LIN {X 0,Y 538.147,Z 457.446,A -85,B 0,C 180,E1 -4137.754,E2 -4137.754} C_VEL
LIN {X 0,Y 538.174,Z 457.449,A -85,B 0,C 180,E1 -4140.748,E2 -4140.748} C_VEL
LIN {X 0,Y 538.129,Z 457.451,A -85,B 0,C 180,E1 -4142.994,E2 -4142.994} C_VEL
LIN {X 0,Y 538.104,Z 457.452,A -85,B 0,C 180,E1 -4145.997,E2 -4145.997} C_VEL
LIN {X 0,Y 538.063,Z 457.459,A -85,B 0,C 180,E1 -4149.017,E2 -4149.017} C_VEL
LIN {X 0,Y 538.07,Z 457.457,A -85,B 0,C 180,E1 -4152.063,E2 -4152.063} C_VEL
LIN {X 0,Y 538.031,Z 457.462,A -85,B 0,C 180,E1 -4155.144,E2 -4155.144} C_VEL
LIN {X 0,Y 538.019,Z 457.465,A -85,B 0,C 180,E1 -4158.27,E2 -4158.27} C_VEL
LIN {X 0,Y 538.029,Z 457.469,A -85,B 0,C 180,E1 -4160.651,E2 -4160.651} C_VEL
LIN {X 0,Y 538.01,Z 457.462,A -85,B 0,C 180,E1 -4163.888,E2 -4163.888} C_VEL
LIN {X 0,Y 538.029,Z 457.464,A -85,B 0,C 180,E1 -4166.367,E2 -4166.367} C_VEL
LIN {X 0,Y 538.019,Z 457.468,A -85,B 0,C 180,E1 -4168.934,E2 -4168.934} C_VEL
LIN {X 0,Y 538.014,Z 457.462,A -85,B 0,C 180,E1 -4171.891,E2 -4171.891} C_VEL
LIN {X 0,Y 538.022,Z 457.468,A -85,B 0,C 180,E1 -4174.622,E2 -4174.622} C_VEL
LIN {X 0,Y 537.995,Z 457.468,A -85,B 0,C 180,E1 -4177.171,E2 -4177.171} C_VEL
LIN {X 0,Y 538.01,Z 457.464,A -85,B 0,C 180,E1 -4180.28,E2 -4180.28} C_VEL
LIN {X 0,Y 537.361,Z 457.552,A -85,B 0,C 180,E1 -4180.906,E2 -4180.906} C_VEL
LIN {X 0,Y 534.511,Z 457.907,A -85,B 0,C 180,E1 -4181.921,E2 -4181.921} C_VEL
LIN {X 0,Y 532.086,Z 458.208,A -85,B 0,C 180,E1 -4182.738,E2 -4182.738} C_VEL
LIN {X 0,Y 531.039,Z 458.333,A -85,B 0,C 180,E1 -4183.369,E2 -4183.369} C_VEL
LIN {X 0,Y 530.951,Z 458.342,A -85,B 0,C 180,E1 -4183.583,E2 -4183.583} C_VEL
LIN {X 0,Y 530.957,Z 458.345,A -85,B 0,C 180,E1 -4186.507,E2 -4186.507} C_VEL
LIN {X 0,Y 531,Z 458.337,A -85,B 0,C 180,E1 -4189.571,E2 -4189.571} C_VEL
LIN {X 0,Y 530.959,Z 458.345,A -85,B 0,C 180,E1 -4192.578,E2 -4192.578} C_VEL
LIN {X 0,Y 530.988,Z 458.341,A -85,B 0,C 180,E1 -4195.312,E2 -4195.312} C_VEL
LIN {X 0,Y 530.975,Z 458.339,A -85,B 0,C 180,E1 -4198.034,E2 -4198.034} C_VEL
LIN {X 0,Y 530.982,Z 458.346,A -85,B 0,C 180,E1 -4200.875,E2 -4200.875} C_VEL
LIN {X 0,Y 530.999,Z 458.341,A -85,B 0,C 180,E1 -4203.258,E2 -4203.258} C_VEL
LIN {X 0,Y 530.991,Z 458.337,A -85,B 0,C 180,E1 -4205.959,E2 -4205.959} C_VEL
LIN {X 0,Y 530.995,Z 458.346,A -85,B 0,C 180,E1 -4209.063,E2 -4209.063} C_VEL
LIN {X 0,Y 531.012,Z 458.334,A -85,B 0,C 180,E1 -4212.279,E2 -4212.279} C_VEL
LIN {X 0,Y 531.015,Z 458.338,A -85,B 0,C 180,E1 -4215.437,E2 -4215.437} C_VEL
LIN {X 0,Y 531.034,Z 458.333,A -85,B 0,C 180,E1 -4218.551,E2 -4218.551} C_VEL
LIN {X 0,Y 531.055,Z 458.333,A -85,B 0,C 180,E1 -4221.631,E2 -4221.631} C_VEL
LIN {X 0,Y 531.123,Z 458.325,A -85,B 0,C 180,E1 -4224.687,E2 -4224.687} C_VEL
LIN {X 0,Y 531.14,Z 458.326,A -85,B 0,C 180,E1 -4227.726,E2 -4227.726} C_VEL
LIN {X 0,Y 531.154,Z 458.469,A -85,B 0,C 180,E1 -4229.338,E2 -4229.338} C_VEL
LIN {X 0,Y 531.34,Z 459.417,A -85,B 0,C 180,E1 -4229.468,E2 -4229.468} C_VEL
LIN {X 0,Y 532.879,Z 464.186,A -85,B 0,C 180,E1 -4229.594,E2 -4229.594} C_VEL
LIN {X 0,Y 532.611,Z 538.316,A -85,B 0,C 180,E1 -4230.616,E2 -4230.616} C_VEL
LIN {X 0,Y 532.49,Z 551.533,A -85,B 0,C 180,E1 -4230.947,E2 -4230.947} C_VEL
LIN {X 0,Y 532.337,Z 564.103,A -85,B 0,C 180,E1 -4231.42,E2 -4231.42} C_VEL
LIN {X 0,Y 532.188,Z 575.279,A -85,B 0,C 180,E1 -4231.988,E2 -4231.988} C_VEL
LIN {X 0,Y 531.934,Z 586.81,A -85,B 0,C 180,E1 -4232.746,E2 -4232.746} C_VEL
LIN {X 0,Y 531.673,Z 597.145,A -85,B 0,C 180,E1 -4233.601,E2 -4233.601} C_VEL
LIN {X 0,Y 531.464,Z 606.464,A -85,B 0,C 180,E1 -4234.552,E2 -4234.552} C_VEL
LIN {X 0,Y 531.243,Z 614.125,A -85,B 0,C 180,E1 -4235.505,E2 -4235.505} C_VEL
LIN {X 0,Y 531.124,Z 621.981,A -85,B 0,C 180,E1 -4236.719,E2 -4236.719} C_VEL
LIN {X 0,Y 530.919,Z 628.515,A -85,B 0,C 180,E1 -4237.991,E2 -4237.991} C_VEL
LIN {X 0,Y 530.782,Z 633.124,A -85,B 0,C 180,E1 -4239.144,E2 -4239.144} C_VEL
LIN {X 0,Y 530.739,Z 635.579,A -85,B 0,C 180,E1 -4239.914,E2 -4239.914} C_VEL
LIN {X 0,Y 530.714,Z 637.565,A -85,B 0,C 180,E1 -4240.685,E2 -4240.685} C_VEL
LIN {X 0,Y 530.683,Z 639.182,A -85,B 0,C 180,E1 -4241.479,E2 -4241.479} C_VEL
LIN {X 0,Y 530.641,Z 640.32,A -85,B 0,C 180,E1 -4242.235,E2 -4242.235} C_VEL
LIN {X 0,Y 530.615,Z 641.044,A -85,B 0,C 180,E1 -4243.014,E2 -4243.014} C_VEL
LIN {X 0,Y 530.608,Z 641.331,A -85,B 0,C 180,E1 -4244.577,E2 -4244.577} C_VEL
LIN {X 0,Y 530.577,Z 640.852,A -85,B 0,C 180,E1 -4245.363,E2 -4245.363} C_VEL
LIN {X 0,Y 530.612,Z 639.937,A -85,B 0,C 180,E1 -4246.151,E2 -4246.151} C_VEL
LIN {X 0,Y 530.707,Z 637.291,A -85,B 0,C 180,E1 -4247.547,E2 -4247.547} C_VEL
LIN {X 0,Y 530.807,Z 633.252,A -85,B 0,C 180,E1 -4248.93,E2 -4248.93} C_VEL
LIN {X 0,Y 530.935,Z 628.451,A -85,B 0,C 180,E1 -4250.132,E2 -4250.132} C_VEL
LIN {X 0,Y 531.091,Z 622.266,A -85,B 0,C 180,E1 -4251.342,E2 -4251.342} C_VEL
LIN {X 0,Y 531.274,Z 614.428,A -85,B 0,C 180,E1 -4252.56,E2 -4252.56} C_VEL
LIN {X 0,Y 531.468,Z 606.223,A -85,B 0,C 180,E1 -4253.58,E2 -4253.58} C_VEL
LIN {X 0,Y 531.699,Z 596.027,A -85,B 0,C 180,E1 -4254.606,E2 -4254.606} C_VEL
LIN {X 0,Y 531.95,Z 585.852,A -85,B 0,C 180,E1 -4255.43,E2 -4255.43} C_VEL
LIN {X 0,Y 532.23,Z 575.243,A -85,B 0,C 180,E1 -4256.114,E2 -4256.114} C_VEL
LIN {X 0,Y 532.362,Z 563.06,A -85,B 0,C 180,E1 -4256.724,E2 -4256.724} C_VEL
LIN {X 0,Y 532.522,Z 551.021,A -85,B 0,C 180,E1 -4257.166,E2 -4257.166} C_VEL
LIN {X 0,Y 532.6,Z 538.195,A -85,B 0,C 180,E1 -4257.481,E2 -4257.481} C_VEL
LIN {X 0,Y 532.82,Z 464.104,A -85,B 0,C 180,E1 -4258.503,E2 -4258.503} C_VEL
LIN {X 0,Y 531.186,Z 459.162,A -85,B 0,C 180,E1 -4258.647,E2 -4258.647} C_VEL
LIN {X 0,Y 531.032,Z 458.389,A -85,B 0,C 180,E1 -4258.816,E2 -4258.816} C_VEL
LIN {X 0,Y 530.968,Z 458.343,A -85,B 0,C 180,E1 -4262.101,E2 -4262.101} C_VEL
LIN {X 0,Y 530.972,Z 458.347,A -85,B 0,C 180,E1 -4264.852,E2 -4264.852} C_VEL
LIN {X 0,Y 530.969,Z 458.342,A -85,B 0,C 180,E1 -4267.509,E2 -4267.509} C_VEL
LIN {X 0,Y 530.984,Z 458.341,A -85,B 0,C 180,E1 -4270.434,E2 -4270.434} C_VEL
LIN {X 0,Y 530.965,Z 458.345,A -85,B 0,C 180,E1 -4273.282,E2 -4273.282} C_VEL
LIN {X 0,Y 530.98,Z 458.34,A -85,B 0,C 180,E1 -4275.623,E2 -4275.623} C_VEL
LIN {X 0,Y 530.998,Z 458.344,A -85,B 0,C 180,E1 -4278.565,E2 -4278.565} C_VEL
LIN {X 0,Y 530.959,Z 458.345,A -85,B 0,C 180,E1 -4281.53,E2 -4281.53} C_VEL
LIN {X 0,Y 531.013,Z 458.494,A -85,B 0,C 180,E1 -4283.121,E2 -4283.121} C_VEL
LIN {X 0,Y 532.299,Z 465.347,A -85,B 0,C 180,E1 -4284.251,E2 -4284.251} C_VEL
LIN {X 0,Y 532.076,Z 480.188,A -85,B 0,C 180,E1 -4286.533,E2 -4286.533} C_VEL
LIN {X 0,Y 531.799,Z 496.041,A -85,B 0,C 180,E1 -4288.976,E2 -4288.976} C_VEL
LIN {X 0,Y 531.405,Z 515.414,A -85,B 0,C 180,E1 -4291.956,E2 -4291.956} C_VEL
LIN {X 0,Y 531.438,Z 516.598,A -85,B 0,C 180,E1 -4292.085,E2 -4292.085} C_VEL
LIN {X 0,Y 532.822,Z 525.632,A -85,B 0,C 180,E1 -4292.271,E2 -4292.271} C_VEL
LIN {X 0,Y 532.386,Z 623.86,A -85,B 0,C 180,E1 -4293.626,E2 -4293.626} C_VEL
LIN {X 0,Y 532.22,Z 636.845,A -85,B 0,C 180,E1 -4293.939,E2 -4293.939} C_VEL
LIN {X 0,Y 531.966,Z 649.489,A -85,B 0,C 180,E1 -4294.415,E2 -4294.415} C_VEL
LIN {X 0,Y 531.828,Z 658.876,A -85,B 0,C 180,E1 -4294.88,E2 -4294.88} C_VEL
LIN {X 0,Y 531.583,Z 668.915,A -85,B 0,C 180,E1 -4295.493,E2 -4295.493} C_VEL
LIN {X 0,Y 531.331,Z 679.721,A -85,B 0,C 180,E1 -4296.311,E2 -4296.311} C_VEL
LIN {X 0,Y 531.076,Z 689.307,A -85,B 0,C 180,E1 -4297.227,E2 -4297.227} C_VEL
LIN {X 0,Y 530.911,Z 696.74,A -85,B 0,C 180,E1 -4298.076,E2 -4298.076} C_VEL
LIN {X 0,Y 530.749,Z 703.942,A -85,B 0,C 180,E1 -4299.052,E2 -4299.052} C_VEL
LIN {X 0,Y 530.621,Z 711.826,A -85,B 0,C 180,E1 -4300.386,E2 -4300.386} C_VEL
LIN {X 0,Y 530.532,Z 716.823,A -85,B 0,C 180,E1 -4301.463,E2 -4301.463} C_VEL
LIN {X 0,Y 530.455,Z 720.818,A -85,B 0,C 180,E1 -4302.543,E2 -4302.543} C_VEL
LIN {X 0,Y 530.373,Z 724.434,A -85,B 0,C 180,E1 -4303.843,E2 -4303.843} C_VEL
LIN {X 0,Y 530.349,Z 726.929,A -85,B 0,C 180,E1 -4305.326,E2 -4305.326} C_VEL
LIN {X 0,Y 530.395,Z 727.726,A -85,B 0,C 180,E1 -4306.202,E2 -4306.202} C_VEL
LIN {X 0,Y 530.368,Z 727.993,A -85,B 0,C 180,E1 -4306.982,E2 -4306.982} C_VEL
LIN {X 0,Y 530.426,Z 727.165,A -85,B 0,C 180,E1 -4308.537,E2 -4308.537} C_VEL
LIN {X 0,Y 530.418,Z 726.192,A -85,B 0,C 180,E1 -4309.31,E2 -4309.31} C_VEL
LIN {X 0,Y 530.406,Z 724.81,A -85,B 0,C 180,E1 -4310.081,E2 -4310.081} C_VEL
LIN {X 0,Y 530.466,Z 721.838,A -85,B 0,C 180,E1 -4311.237,E2 -4311.237} C_VEL
LIN {X 0,Y 530.53,Z 717.804,A -85,B 0,C 180,E1 -4312.388,E2 -4312.388} C_VEL
LIN {X 0,Y 530.594,Z 712.072,A -85,B 0,C 180,E1 -4313.655,E2 -4313.655} C_VEL
LIN {X 0,Y 530.65,Z 705.099,A -85,B 0,C 180,E1 -4314.871,E2 -4314.871} C_VEL
LIN {X 0,Y 530.87,Z 696.79,A -85,B 0,C 180,E1 -4316.015,E2 -4316.015} C_VEL
LIN {X 0,Y 531.103,Z 688.364,A -85,B 0,C 180,E1 -4316.966,E2 -4316.966} C_VEL
LIN {X 0,Y 531.388,Z 678.035,A -85,B 0,C 180,E1 -4317.916,E2 -4317.916} C_VEL
LIN {X 0,Y 531.55,Z 669.189,A -85,B 0,C 180,E1 -4318.58,E2 -4318.58} C_VEL
LIN {X 0,Y 531.763,Z 660.023,A -85,B 0,C 180,E1 -4319.148,E2 -4319.148} C_VEL
LIN {X 0,Y 532.007,Z 649.602,A -85,B 0,C 180,E1 -4319.669,E2 -4319.669} C_VEL
LIN {X 0,Y 532.27,Z 636.266,A -85,B 0,C 180,E1 -4320.166,E2 -4320.166} C_VEL
LIN {X 0,Y 532.365,Z 624.629,A -85,B 0,C 180,E1 -4320.449,E2 -4320.449} C_VEL
LIN {X 0,Y 532.735,Z 558.302,A -85,B 0,C 180,E1 -4321.37,E2 -4321.37} C_VEL
LIN {X 0,Y 532.648,Z 524.275,A -85,B 0,C 180,E1 -4321.843,E2 -4321.843} C_VEL
LIN {X 0,Y 531.495,Z 517.058,A -85,B 0,C 180,E1 -4321.989,E2 -4321.989} C_VEL
LIN {X 0,Y 531.446,Z 515.98,A -85,B 0,C 180,E1 -4322.084,E2 -4322.084} C_VEL
LIN {X 0,Y 531.728,Z 499.989,A -85,B 0,C 180,E1 -4324.549,E2 -4324.549} C_VEL
LIN {X 0,Y 532.052,Z 481.832,A -85,B 0,C 180,E1 -4327.308,E2 -4327.308} C_VEL
LIN {X 0,Y 532.261,Z 465.964,A -85,B 0,C 180,E1 -4329.692,E2 -4329.692} C_VEL
LIN {X 0,Y 531.057,Z 458.412,A -85,B 0,C 180,E1 -4330.895,E2 -4330.895} C_VEL
LIN {X 0,Y 530.96,Z 458.346,A -85,B 0,C 180,E1 -4333.784,E2 -4333.784} C_VEL
LIN {X 0,Y 530.97,Z 458.342,A -85,B 0,C 180,E1 -4336.139,E2 -4336.139} C_VEL
LIN {X 0,Y 530.978,Z 458.343,A -85,B 0,C 180,E1 -4338.522,E2 -4338.522} C_VEL
LIN {X 0,Y 531.005,Z 458.344,A -85,B 0,C 180,E1 -4340.938,E2 -4340.938} C_VEL
LIN {X 0,Y 530.963,Z 458.343,A -85,B 0,C 180,E1 -4344.226,E2 -4344.226} C_VEL
LIN {X 0,Y 531.005,Z 458.344,A -85,B 0,C 180,E1 -4346.744,E2 -4346.744} C_VEL
LIN {X 0,Y 530.989,Z 458.341,A -85,B 0,C 180,E1 -4349.322,E2 -4349.322} C_VEL
LIN {X 0,Y 530.974,Z 458.341,A -85,B 0,C 180,E1 -4352.1,E2 -4352.1} C_VEL
LIN {X 0,Y 530.979,Z 458.346,A -85,B 0,C 180,E1 -4354.851,E2 -4354.851} C_VEL
LIN {X 0,Y 530.973,Z 458.341,A -85,B 0,C 180,E1 -4357.507,E2 -4357.507} C_VEL
LIN {X 0,Y 530.989,Z 458.345,A -85,B 0,C 180,E1 -4360.433,E2 -4360.433} C_VEL
LIN {X 0,Y 530.968,Z 458.342,A -85,B 0,C 180,E1 -4363.281,E2 -4363.281} C_VEL
LIN {X 0,Y 530.984,Z 458.34,A -85,B 0,C 180,E1 -4365.622,E2 -4365.622} C_VEL
LIN {X 0,Y 531.001,Z 458.344,A -85,B 0,C 180,E1 -4368.564,E2 -4368.564} C_VEL
LIN {X 0,Y 530.961,Z 458.337,A -85,B 0,C 180,E1 -4371.528,E2 -4371.528} C_VEL
LIN {X 0,Y 530.954,Z 458.347,A -85,B 0,C 180,E1 -4374.379,E2 -4374.379} C_VEL
LIN {X 0,Y 530.973,Z 458.343,A -85,B 0,C 180,E1 -4377.133,E2 -4377.133} C_VEL
LIN {X 0,Y 530.966,Z 458.348,A -85,B 0,C 180,E1 -4379.802,E2 -4379.802} C_VEL
LIN {X 0,Y 531.03,Z 458.561,A -85,B 0,C 180,E1 -4381.7,E2 -4381.7} C_VEL
LIN {X 0,Y 533.429,Z 469.801,A -85,B 0,C 180,E1 -4383.175,E2 -4383.175} C_VEL
LIN {X 0,Y 533.157,Z 486.764,A -85,B 0,C 180,E1 -4385.18,E2 -4385.18} C_VEL
LIN {X 0,Y 532.709,Z 508.501,A -85,B 0,C 180,E1 -4387.709,E2 -4387.709} C_VEL
LIN {X 0,Y 532.341,Z 529.733,A -85,B 0,C 180,E1 -4390.125,E2 -4390.125} C_VEL
LIN {X 0,Y 531.921,Z 556.102,A -85,B 0,C 180,E1 -4393.1,E2 -4393.1} C_VEL
LIN {X 0,Y 531.697,Z 573.392,A -85,B 0,C 180,E1 -4395.022,E2 -4395.022} C_VEL
LIN {X 0,Y 532.816,Z 582.327,A -85,B 0,C 180,E1 -4395.188,E2 -4395.188} C_VEL
LIN {X 0,Y 532.437,Z 683.75,A -85,B 0,C 180,E1 -4396.57,E2 -4396.57} C_VEL
LIN {X 0,Y 532.271,Z 696.373,A -85,B 0,C 180,E1 -4396.882,E2 -4396.882} C_VEL
LIN {X 0,Y 532.045,Z 709.34,A -85,B 0,C 180,E1 -4397.361,E2 -4397.361} C_VEL
LIN {X 0,Y 531.811,Z 721.287,A -85,B 0,C 180,E1 -4397.966,E2 -4397.966} C_VEL
LIN {X 0,Y 531.521,Z 733.176,A -85,B 0,C 180,E1 -4398.752,E2 -4398.752} C_VEL
LIN {X 0,Y 531.285,Z 743.591,A -85,B 0,C 180,E1 -4399.615,E2 -4399.615} C_VEL
LIN {X 0,Y 531.063,Z 752.102,A -85,B 0,C 180,E1 -4400.477,E2 -4400.477} C_VEL
LIN {X 0,Y 530.886,Z 759.951,A -85,B 0,C 180,E1 -4401.434,E2 -4401.434} C_VEL
LIN {X 0,Y 530.686,Z 767.614,A -85,B 0,C 180,E1 -4402.58,E2 -4402.58} C_VEL
LIN {X 0,Y 530.605,Z 774.674,A -85,B 0,C 180,E1 -4403.916,E2 -4403.916} C_VEL
LIN {X 0,Y 530.459,Z 779.368,A -85,B 0,C 180,E1 -4405.058,E2 -4405.058} C_VEL
LIN {X 0,Y 530.516,Z 782.954,A -85,B 0,C 180,E1 -4406.201,E2 -4406.201} C_VEL
LIN {X 0,Y 530.457,Z 784.804,A -85,B 0,C 180,E1 -4406.961,E2 -4406.961} C_VEL
LIN {X 0,Y 530.411,Z 786.192,A -85,B 0,C 180,E1 -4407.721,E2 -4407.721} C_VEL
LIN {X 0,Y 530.344,Z 787.785,A -85,B 0,C 180,E1 -4409.239,E2 -4409.239} C_VEL
LIN {X 0,Y 530.342,Z 788,A -85,B 0,C 180,E1 -4409.999,E2 -4409.999} C_VEL
LIN {X 0,Y 530.361,Z 787.185,A -85,B 0,C 180,E1 -4411.517,E2 -4411.517} C_VEL
LIN {X 0,Y 530.411,Z 786.198,A -85,B 0,C 180,E1 -4412.277,E2 -4412.277} C_VEL
LIN {X 0,Y 530.457,Z 784.813,A -85,B 0,C 180,E1 -4413.037,E2 -4413.037} C_VEL
LIN {X 0,Y 530.522,Z 781.899,A -85,B 0,C 180,E1 -4414.177,E2 -4414.177} C_VEL
LIN {X 0,Y 530.524,Z 777.953,A -85,B 0,C 180,E1 -4415.319,E2 -4415.319} C_VEL
LIN {X 0,Y 530.594,Z 772.289,A -85,B 0,C 180,E1 -4416.577,E2 -4416.577} C_VEL
LIN {X 0,Y 530.757,Z 765.244,A -85,B 0,C 180,E1 -4417.799,E2 -4417.799} C_VEL
LIN {X 0,Y 530.929,Z 757.003,A -85,B 0,C 180,E1 -4418.947,E2 -4418.947} C_VEL
LIN {X 0,Y 531.141,Z 748.553,A -85,B 0,C 180,E1 -4419.904,E2 -4419.904} C_VEL
LIN {X 0,Y 531.409,Z 738.107,A -85,B 0,C 180,E1 -4420.861,E2 -4420.861} C_VEL
LIN {X 0,Y 531.701,Z 727.156,A -85,B 0,C 180,E1 -4421.669,E2 -4421.669} C_VEL
LIN {X 0,Y 531.929,Z 716.429,A -85,B 0,C 180,E1 -4422.3,E2 -4422.3} C_VEL
LIN {X 0,Y 532.113,Z 704.795,A -85,B 0,C 180,E1 -4422.828,E2 -4422.828} C_VEL
LIN {X 0,Y 532.3,Z 692.228,A -85,B 0,C 180,E1 -4423.236,E2 -4423.236} C_VEL
LIN {X 0,Y 532.475,Z 679.523,A -85,B 0,C 180,E1 -4423.499,E2 -4423.499} C_VEL
LIN {X 0,Y 532.716,Z 581.48,A -85,B 0,C 180,E1 -4424.827,E2 -4424.827} C_VEL
LIN {X 0,Y 531.714,Z 573.469,A -85,B 0,C 180,E1 -4424.976,E2 -4424.976} C_VEL
LIN {X 0,Y 532.086,Z 546.475,A -85,B 0,C 180,E1 -4428.009,E2 -4428.009} C_VEL
LIN {X 0,Y 532.603,Z 517.827,A -85,B 0,C 180,E1 -4431.275,E2 -4431.275} C_VEL
LIN {X 0,Y 533.136,Z 491.898,A -85,B 0,C 180,E1 -4434.281,E2 -4434.281} C_VEL
LIN {X 0,Y 533.53,Z 470.521,A -85,B 0,C 180,E1 -4436.817,E2 -4436.817} C_VEL
LIN {X 0,Y 531.021,Z 458.46,A -85,B 0,C 180,E1 -4438.428,E2 -4438.428} C_VEL
LIN {X 0,Y 530.946,Z 458.346,A -85,B 0,C 180,E1 -4441.078,E2 -4441.078} C_VEL
LIN {X 0,Y 530.95,Z 458.349,A -85,B 0,C 180,E1 -4443.774,E2 -4443.774} C_VEL
LIN {X 0,Y 530.928,Z 458.348,A -85,B 0,C 180,E1 -4446.559,E2 -4446.559} C_VEL
LIN {X 0,Y 530.96,Z 458.341,A -85,B 0,C 180,E1 -4449.444,E2 -4449.444} C_VEL
LIN {X 0,Y 530.923,Z 458.351,A -85,B 0,C 180,E1 -4452.46,E2 -4452.46} C_VEL
LIN {X 0,Y 530.962,Z 458.341,A -85,B 0,C 180,E1 -4455.45,E2 -4455.45} C_VEL
LIN {X 0,Y 530.969,Z 458.344,A -85,B 0,C 180,E1 -4458.562,E2 -4458.562} C_VEL
LIN {X 0,Y 530.942,Z 458.343,A -85,B 0,C 180,E1 -4461.528,E2 -4461.528} C_VEL
LIN {X 0,Y 530.939,Z 458.352,A -85,B 0,C 180,E1 -4464.378,E2 -4464.378} C_VEL
LIN {X 0,Y 530.956,Z 458.341,A -85,B 0,C 180,E1 -4467.132,E2 -4467.132} C_VEL
LIN {X 0,Y 530.948,Z 458.344,A -85,B 0,C 180,E1 -4469.801,E2 -4469.801} C_VEL
LIN {X 0,Y 530.996,Z 458.344,A -85,B 0,C 180,E1 -4472.467,E2 -4472.467} C_VEL
LIN {X 0,Y 530.96,Z 458.342,A -85,B 0,C 180,E1 -4474.94,E2 -4474.94} C_VEL
LIN {X 0,Y 530.963,Z 458.343,A -85,B 0,C 180,E1 -4477.897,E2 -4477.897} C_VEL
LIN {X 0,Y 530.97,Z 458.345,A -85,B 0,C 180,E1 -4480.676,E2 -4480.676} C_VEL
LIN {X 0,Y 530.966,Z 458.341,A -85,B 0,C 180,E1 -4483.07,E2 -4483.07} C_VEL
LIN {X 0,Y 531,Z 458.336,A -85,B 0,C 180,E1 -4485.435,E2 -4485.435} C_VEL
LIN {X 0,Y 531.034,Z 458.34,A -85,B 0,C 180,E1 -4488.549,E2 -4488.549} C_VEL
LIN {X 0,Y 531.037,Z 458.331,A -85,B 0,C 180,E1 -4491.629,E2 -4491.629} C_VEL
LIN {X 0,Y 531.102,Z 458.33,A -85,B 0,C 180,E1 -4494.685,E2 -4494.685} C_VEL
LIN {X 0,Y 531.12,Z 458.321,A -85,B 0,C 180,E1 -4497.725,E2 -4497.725} C_VEL
LIN {X 0,Y 531.143,Z 458.324,A -85,B 0,C 180,E1 -4500.758,E2 -4500.758} C_VEL
LIN {X 0,Y 531.095,Z 458.327,A -85,B 0,C 180,E1 -4503.034,E2 -4503.034} C_VEL
LIN {X 0,Y 531.06,Z 458.33,A -85,B 0,C 180,E1 -4506.077,E2 -4506.077} C_VEL
LIN {X 0,Y 531.046,Z 458.336,A -85,B 0,C 180,E1 -4508.37,E2 -4508.37} C_VEL
LIN {X 0,Y 531.044,Z 458.33,A -85,B 0,C 180,E1 -4511.676,E2 -4511.676} C_VEL
LIN {X 0,Y 531.016,Z 458.339,A -85,B 0,C 180,E1 -4514.956,E2 -4514.956} C_VEL
LIN {X 0,Y 531.002,Z 458.335,A -85,B 0,C 180,E1 -4517.723,E2 -4517.723} C_VEL
LIN {X 0,Y 530.988,Z 458.343,A -85,B 0,C 180,E1 -4520.938,E2 -4520.938} C_VEL
LIN {X 0,Y 530.966,Z 458.342,A -85,B 0,C 180,E1 -4524.225,E2 -4524.225} C_VEL
LIN {X 0,Y 530.993,Z 458.347,A -85,B 0,C 180,E1 -4526.744,E2 -4526.744} C_VEL
LIN {X 0,Y 530.969,Z 458.341,A -85,B 0,C 180,E1 -4529.323,E2 -4529.323} C_VEL
LIN {X 0,Y 530.967,Z 458.341,A -85,B 0,C 180,E1 -4532.104,E2 -4532.104} C_VEL
LIN {X 0,Y 530.978,Z 458.347,A -85,B 0,C 180,E1 -4534.855,E2 -4534.855} C_VEL
LIN {X 0,Y 530.954,Z 458.342,A -85,B 0,C 180,E1 -4537.508,E2 -4537.508} C_VEL
LIN {X 0,Y 530.973,Z 458.342,A -85,B 0,C 180,E1 -4540.433,E2 -4540.433} C_VEL
LIN {X 0,Y 530.959,Z 458.344,A -85,B 0,C 180,E1 -4543.283,E2 -4543.283} C_VEL
LIN {X 0,Y 530.951,Z 458.342,A -85,B 0,C 180,E1 -4543.583,E2 -4543.583} C_VEL
LIN {X 0,Y 530.279,Z 458.427,A -85,B 0,C 180,E1 -4544.216,E2 -4544.216} C_VEL
LIN {X 0,Y 527.431,Z 458.789,A -85,B 0,C 180,E1 -4545.245,E2 -4545.245} C_VEL
LIN {X 0,Y 525.029,Z 459.093,A -85,B 0,C 180,E1 -4546.074,E2 -4546.074} C_VEL
LIN {X 0,Y 523.998,Z 459.218,A -85,B 0,C 180,E1 -4546.713,E2 -4546.713} C_VEL
LIN {X 0,Y 523.914,Z 459.226,A -85,B 0,C 180,E1 -4546.93,E2 -4546.93} C_VEL
LIN {X 0,Y 523.968,Z 459.211,A -85,B 0,C 180,E1 -4549.924,E2 -4549.924} C_VEL
LIN {X 0,Y 523.901,Z 459.229,A -85,B 0,C 180,E1 -4552.869,E2 -4552.869} C_VEL
LIN {X 0,Y 523.932,Z 459.217,A -85,B 0,C 180,E1 -4555.712,E2 -4555.712} C_VEL
LIN {X 0,Y 523.924,Z 459.219,A -85,B 0,C 180,E1 -4558.458,E2 -4558.458} C_VEL
LIN {X 0,Y 523.933,Z 459.224,A -85,B 0,C 180,E1 -4561.127,E2 -4561.127} C_VEL
LIN {X 0,Y 523.977,Z 459.21,A -85,B 0,C 180,E1 -4563.981,E2 -4563.981} C_VEL
LIN {X 0,Y 523.93,Z 459.217,A -85,B 0,C 180,E1 -4566.272,E2 -4566.272} C_VEL
LIN {X 0,Y 523.941,Z 459.22,A -85,B 0,C 180,E1 -4568.768,E2 -4568.768} C_VEL
LIN {X 0,Y 523.947,Z 459.221,A -85,B 0,C 180,E1 -4571.222,E2 -4571.222} C_VEL
LIN {X 0,Y 523.934,Z 459.218,A -85,B 0,C 180,E1 -4573.64,E2 -4573.64} C_VEL
LIN {X 0,Y 523.937,Z 459.215,A -85,B 0,C 180,E1 -4576.029,E2 -4576.029} C_VEL
LIN {X 0,Y 524.009,Z 459.207,A -85,B 0,C 180,E1 -4578.395,E2 -4578.395} C_VEL
LIN {X 0,Y 524.003,Z 459.213,A -85,B 0,C 180,E1 -4581.517,E2 -4581.517} C_VEL
LIN {X 0,Y 524.084,Z 459.202,A -85,B 0,C 180,E1 -4584.615,E2 -4584.615} C_VEL
LIN {X 0,Y 524.112,Z 459.202,A -85,B 0,C 180,E1 -4587.696,E2 -4587.696} C_VEL
LIN {X 0,Y 524.107,Z 459.353,A -85,B 0,C 180,E1 -4589.137,E2 -4589.137} C_VEL
LIN {X 0,Y 524.331,Z 460.326,A -85,B 0,C 180,E1 -4589.269,E2 -4589.269} C_VEL
LIN {X 0,Y 526.005,Z 465.293,A -85,B 0,C 180,E1 -4589.403,E2 -4589.403} C_VEL
LIN {X 0,Y 525.723,Z 540.189,A -85,B 0,C 180,E1 -4590.456,E2 -4590.456} C_VEL
LIN {X 0,Y 525.639,Z 553.033,A -85,B 0,C 180,E1 -4590.791,E2 -4590.791} C_VEL
LIN {X 0,Y 525.454,Z 566.022,A -85,B 0,C 180,E1 -4591.295,E2 -4591.295} C_VEL
LIN {X 0,Y 525.268,Z 577.726,A -85,B 0,C 180,E1 -4591.918,E2 -4591.918} C_VEL
LIN {X 0,Y 525.022,Z 588.944,A -85,B 0,C 180,E1 -4592.687,E2 -4592.687} C_VEL
LIN {X 0,Y 524.721,Z 599.09,A -85,B 0,C 180,E1 -4593.553,E2 -4593.553} C_VEL
LIN {X 0,Y 524.528,Z 607.374,A -85,B 0,C 180,E1 -4594.42,E2 -4594.42} C_VEL
LIN {X 0,Y 524.286,Z 615.049,A -85,B 0,C 180,E1 -4595.385,E2 -4595.385} C_VEL
LIN {X 0,Y 524.167,Z 622.52,A -85,B 0,C 180,E1 -4596.545,E2 -4596.545} C_VEL
LIN {X 0,Y 523.953,Z 628.568,A -85,B 0,C 180,E1 -4597.71,E2 -4597.71} C_VEL
LIN {X 0,Y 523.807,Z 633.369,A -85,B 0,C 180,E1 -4598.877,E2 -4598.877} C_VEL
LIN {X 0,Y 523.712,Z 637.067,A -85,B 0,C 180,E1 -4600.048,E2 -4600.048} C_VEL
LIN {X 0,Y 523.651,Z 640.36,A -85,B 0,C 180,E1 -4601.553,E2 -4601.553} C_VEL
LIN {X 0,Y 523.619,Z 641.492,A -85,B 0,C 180,E1 -4602.402,E2 -4602.402} C_VEL
LIN {X 0,Y 523.55,Z 642.411,A -85,B 0,C 180,E1 -4603.984,E2 -4603.984} C_VEL
LIN {X 0,Y 523.581,Z 642.169,A -85,B 0,C 180,E1 -4604.884,E2 -4604.884} C_VEL
LIN {X 0,Y 523.594,Z 640.651,A -85,B 0,C 180,E1 -4606.373,E2 -4606.373} C_VEL
LIN {X 0,Y 523.721,Z 638.084,A -85,B 0,C 180,E1 -4607.68,E2 -4607.68} C_VEL
LIN {X 0,Y 523.78,Z 634.935,A -85,B 0,C 180,E1 -4608.787,E2 -4608.787} C_VEL
LIN {X 0,Y 523.952,Z 629.836,A -85,B 0,C 180,E1 -4610.126,E2 -4610.126} C_VEL
LIN {X 0,Y 524.115,Z 623.291,A -85,B 0,C 180,E1 -4611.434,E2 -4611.434} C_VEL
LIN {X 0,Y 524.352,Z 615.269,A -85,B 0,C 180,E1 -4612.694,E2 -4612.694} C_VEL
LIN {X 0,Y 524.558,Z 607.271,A -85,B 0,C 180,E1 -4613.701,E2 -4613.701} C_VEL
LIN {X 0,Y 524.805,Z 597.082,A -85,B 0,C 180,E1 -4614.74,E2 -4614.74} C_VEL
LIN {X 0,Y 525.08,Z 586.928,A -85,B 0,C 180,E1 -4615.574,E2 -4615.574} C_VEL
LIN {X 0,Y 525.372,Z 575.256,A -85,B 0,C 180,E1 -4616.328,E2 -4616.328} C_VEL
LIN {X 0,Y 525.508,Z 562.955,A -85,B 0,C 180,E1 -4616.94,E2 -4616.94} C_VEL
LIN {X 0,Y 525.666,Z 550.486,A -85,B 0,C 180,E1 -4617.388,E2 -4617.388} C_VEL
LIN {X 0,Y 525.735,Z 537.836,A -85,B 0,C 180,E1 -4617.681,E2 -4617.681} C_VEL
LIN {X 0,Y 525.927,Z 465.337,A -85,B 0,C 180,E1 -4618.693,E2 -4618.693} C_VEL
LIN {X 0,Y 524.157,Z 460.077,A -85,B 0,C 180,E1 -4618.846,E2 -4618.846} C_VEL
LIN {X 0,Y 523.98,Z 459.308,A -85,B 0,C 180,E1 -4618.987,E2 -4618.987} C_VEL
LIN {X 0,Y 523.924,Z 459.221,A -85,B 0,C 180,E1 -4621.545,E2 -4621.545} C_VEL
LIN {X 0,Y 523.924,Z 459.222,A -85,B 0,C 180,E1 -4624.292,E2 -4624.292} C_VEL
LIN {X 0,Y 523.91,Z 459.225,A -85,B 0,C 180,E1 -4627.133,E2 -4627.133} C_VEL
LIN {X 0,Y 523.942,Z 459.215,A -85,B 0,C 180,E1 -4630.131,E2 -4630.131} C_VEL
LIN {X 0,Y 523.939,Z 459.22,A -85,B 0,C 180,E1 -4632.46,E2 -4632.46} C_VEL
LIN {X 0,Y 523.946,Z 459.219,A -85,B 0,C 180,E1 -4635.311,E2 -4635.311} C_VEL
LIN {X 0,Y 523.96,Z 459.221,A -85,B 0,C 180,E1 -4638.691,E2 -4638.691} C_VEL
LIN {X 0,Y 523.92,Z 459.225,A -85,B 0,C 180,E1 -4641.082,E2 -4641.082} C_VEL
LIN {X 0,Y 523.985,Z 459.405,A -85,B 0,C 180,E1 -4642.968,E2 -4642.968} C_VEL
LIN {X 0,Y 525.355,Z 466.551,A -85,B 0,C 180,E1 -4644.149,E2 -4644.149} C_VEL
LIN {X 0,Y 525.21,Z 478.888,A -85,B 0,C 180,E1 -4646.063,E2 -4646.063} C_VEL
LIN {X 0,Y 524.892,Z 494.782,A -85,B 0,C 180,E1 -4648.521,E2 -4648.521} C_VEL
LIN {X 0,Y 524.482,Z 514.628,A -85,B 0,C 180,E1 -4651.596,E2 -4651.596} C_VEL
LIN {X 0,Y 524.492,Z 517.042,A -85,B 0,C 180,E1 -4651.894,E2 -4651.894} C_VEL
LIN {X 0,Y 525.967,Z 526.584,A -85,B 0,C 180,E1 -4652.087,E2 -4652.087} C_VEL
LIN {X 0,Y 525.473,Z 624.303,A -85,B 0,C 180,E1 -4653.461,E2 -4653.461} C_VEL
LIN {X 0,Y 525.293,Z 637.877,A -85,B 0,C 180,E1 -4653.8,E2 -4653.8} C_VEL
LIN {X 0,Y 525.023,Z 649.958,A -85,B 0,C 180,E1 -4654.265,E2 -4654.265} C_VEL
LIN {X 0,Y 524.839,Z 661.187,A -85,B 0,C 180,E1 -4654.84,E2 -4654.84} C_VEL
LIN {X 0,Y 524.559,Z 672.303,A -85,B 0,C 180,E1 -4655.561,E2 -4655.561} C_VEL
LIN {X 0,Y 524.285,Z 682.393,A -85,B 0,C 180,E1 -4656.393,E2 -4656.393} C_VEL
LIN {X 0,Y 524.063,Z 689.738,A -85,B 0,C 180,E1 -4657.114,E2 -4657.114} C_VEL
LIN {X 0,Y 523.839,Z 698.488,A -85,B 0,C 180,E1 -4658.143,E2 -4658.143} C_VEL
LIN {X 0,Y 523.624,Z 706.883,A -85,B 0,C 180,E1 -4659.371,E2 -4659.371} C_VEL
LIN {X 0,Y 523.54,Z 712.477,A -85,B 0,C 180,E1 -4660.391,E2 -4660.391} C_VEL
LIN {X 0,Y 523.445,Z 717.859,A -85,B 0,C 180,E1 -4661.608,E2 -4661.608} C_VEL
LIN {X 0,Y 523.358,Z 722.011,A -85,B 0,C 180,E1 -4662.817,E2 -4662.817} C_VEL
LIN {X 0,Y 523.283,Z 724.07,A -85,B 0,C 180,E1 -4663.618,E2 -4663.618} C_VEL
LIN {X 0,Y 523.247,Z 725.689,A -85,B 0,C 180,E1 -4664.418,E2 -4664.418} C_VEL
LIN {X 0,Y 523.273,Z 726.928,A -85,B 0,C 180,E1 -4665.248,E2 -4665.248} C_VEL
LIN {X 0,Y 523.283,Z 727.693,A -85,B 0,C 180,E1 -4666.01,E2 -4666.01} C_VEL
LIN {X 0,Y 523.285,Z 727.91,A -85,B 0,C 180,E1 -4667.591,E2 -4667.591} C_VEL
LIN {X 0,Y 523.368,Z 727.189,A -85,B 0,C 180,E1 -4668.605,E2 -4668.605} C_VEL
LIN {X 0,Y 523.323,Z 725.214,A -85,B 0,C 180,E1 -4669.946,E2 -4669.946} C_VEL
LIN {X 0,Y 523.369,Z 722.479,A -85,B 0,C 180,E1 -4671.117,E2 -4671.117} C_VEL
LIN {X 0,Y 523.443,Z 718.663,A -85,B 0,C 180,E1 -4672.284,E2 -4672.284} C_VEL
LIN {X 0,Y 523.551,Z 713.954,A -85,B 0,C 180,E1 -4673.397,E2 -4673.397} C_VEL
LIN {X 0,Y 523.606,Z 708.659,A -85,B 0,C 180,E1 -4674.416,E2 -4674.416} C_VEL
LIN {X 0,Y 523.744,Z 702.592,A -85,B 0,C 180,E1 -4675.382,E2 -4675.382} C_VEL
LIN {X 0,Y 523.893,Z 695.368,A -85,B 0,C 180,E1 -4676.347,E2 -4676.347} C_VEL
LIN {X 0,Y 524.179,Z 685.573,A -85,B 0,C 180,E1 -4677.407,E2 -4677.407} C_VEL
LIN {X 0,Y 524.463,Z 675.634,A -85,B 0,C 180,E1 -4678.273,E2 -4678.273} C_VEL
LIN {X 0,Y 524.735,Z 664.783,A -85,B 0,C 180,E1 -4679.041,E2 -4679.041} C_VEL
LIN {X 0,Y 524.986,Z 653.427,A -85,B 0,C 180,E1 -4679.665,E2 -4679.665} C_VEL
LIN {X 0,Y 525.249,Z 641.965,A -85,B 0,C 180,E1 -4680.144,E2 -4680.144} C_VEL
LIN {X 0,Y 525.415,Z 629.155,A -85,B 0,C 180,E1 -4680.527,E2 -4680.527} C_VEL
LIN {X 0,Y 525.571,Z 613.77,A -85,B 0,C 180,E1 -4680.79,E2 -4680.79} C_VEL
LIN {X 0,Y 525.849,Z 525.433,A -85,B 0,C 180,E1 -4682.023,E2 -4682.023} C_VEL
LIN {X 0,Y 524.54,Z 517.063,A -85,B 0,C 180,E1 -4682.208,E2 -4682.208} C_VEL
LIN {X 0,Y 524.71,Z 504.95,A -85,B 0,C 180,E1 -4684.033,E2 -4684.033} C_VEL
LIN {X 0,Y 525.058,Z 485.18,A -85,B 0,C 180,E1 -4687.082,E2 -4687.082} C_VEL
LIN {X 0,Y 525.322,Z 468.156,A -85,B 0,C 180,E1 -4689.627,E2 -4689.627} C_VEL
LIN {X 0,Y 524.441,Z 461.711,A -85,B 0,C 180,E1 -4690.618,E2 -4690.618} C_VEL
LIN {X 0,Y 524.03,Z 459.285,A -85,B 0,C 180,E1 -4691.042,E2 -4691.042} C_VEL
LIN {X 0,Y 523.918,Z 459.223,A -85,B 0,C 180,E1 -4693.973,E2 -4693.973} C_VEL
LIN {X 0,Y 523.915,Z 459.222,A -85,B 0,C 180,E1 -4696.362,E2 -4696.362} C_VEL
LIN {X 0,Y 523.943,Z 459.223,A -85,B 0,C 180,E1 -4698.78,E2 -4698.78} C_VEL
LIN {X 0,Y 523.952,Z 459.222,A -85,B 0,C 180,E1 -4701.233,E2 -4701.233} C_VEL
LIN {X 0,Y 523.943,Z 459.218,A -85,B 0,C 180,E1 -4704.197,E2 -4704.197} C_VEL
LIN {X 0,Y 523.955,Z 459.22,A -85,B 0,C 180,E1 -4707.133,E2 -4707.133} C_VEL
LIN {X 0,Y 523.946,Z 459.216,A -85,B 0,C 180,E1 -4709.756,E2 -4709.756} C_VEL
LIN {X 0,Y 523.942,Z 459.221,A -85,B 0,C 180,E1 -4712.449,E2 -4712.449} C_VEL
LIN {X 0,Y 523.929,Z 459.22,A -85,B 0,C 180,E1 -4715.226,E2 -4715.226} C_VEL
LIN {X 0,Y 523.923,Z 459.221,A -85,B 0,C 180,E1 -4718.102,E2 -4718.102} C_VEL
LIN {X 0,Y 523.947,Z 459.218,A -85,B 0,C 180,E1 -4721.092,E2 -4721.092} C_VEL
LIN {X 0,Y 523.938,Z 459.223,A -85,B 0,C 180,E1 -4724.228,E2 -4724.228} C_VEL
LIN {X 0,Y 523.924,Z 459.222,A -85,B 0,C 180,E1 -4726.832,E2 -4726.832} C_VEL
LIN {X 0,Y 523.947,Z 459.218,A -85,B 0,C 180,E1 -4728.907,E2 -4728.907} C_VEL
LIN {X 0,Y 523.92,Z 459.215,A -85,B 0,C 180,E1 -4731.897,E2 -4731.897} C_VEL
LIN {X 0,Y 523.925,Z 459.217,A -85,B 0,C 180,E1 -4734.912,E2 -4734.912} C_VEL
LIN {X 0,Y 523.942,Z 459.222,A -85,B 0,C 180,E1 -4737.679,E2 -4737.679} C_VEL
LIN {X 0,Y 523.959,Z 459.222,A -85,B 0,C 180,E1 -4740.676,E2 -4740.676} C_VEL
LIN {X 0,Y 523.998,Z 459.46,A -85,B 0,C 180,E1 -4741.497,E2 -4741.497} C_VEL
LIN {X 0,Y 526.569,Z 471.754,A -85,B 0,C 180,E1 -4743.141,E2 -4743.141} C_VEL
LIN {X 0,Y 526.065,Z 495.325,A -85,B 0,C 180,E1 -4745.953,E2 -4745.953} C_VEL
LIN {X 0,Y 525.603,Z 519.967,A -85,B 0,C 180,E1 -4748.836,E2 -4748.836} C_VEL
LIN {X 0,Y 525.058,Z 546.387,A -85,B 0,C 180,E1 -4751.87,E2 -4751.87} C_VEL
LIN {X 0,Y 524.636,Z 572.357,A -85,B 0,C 180,E1 -4754.815,E2 -4754.815} C_VEL
LIN {X 0,Y 525.94,Z 584.263,A -85,B 0,C 180,E1 -4755.03,E2 -4755.03} C_VEL
LIN {X 0,Y 525.548,Z 682.695,A -85,B 0,C 180,E1 -4756.391,E2 -4756.391} C_VEL
LIN {X 0,Y 525.335,Z 695.331,A -85,B 0,C 180,E1 -4756.705,E2 -4756.705} C_VEL
LIN {X 0,Y 525.066,Z 708.392,A -85,B 0,C 180,E1 -4757.191,E2 -4757.191} C_VEL
LIN {X 0,Y 524.836,Z 719.455,A -85,B 0,C 180,E1 -4757.744,E2 -4757.744} C_VEL
LIN {X 0,Y 524.556,Z 731.291,A -85,B 0,C 180,E1 -4758.503,E2 -4758.503} C_VEL
LIN {X 0,Y 524.268,Z 742.128,A -85,B 0,C 180,E1 -4759.377,E2 -4759.377} C_VEL
LIN {X 0,Y 524.029,Z 751.916,A -85,B 0,C 180,E1 -4760.348,E2 -4760.348} C_VEL
LIN {X 0,Y 523.851,Z 759.907,A -85,B 0,C 180,E1 -4761.318,E2 -4761.318} C_VEL
LIN {X 0,Y 523.635,Z 767.614,A -85,B 0,C 180,E1 -4762.479,E2 -4762.479} C_VEL
LIN {X 0,Y 523.516,Z 774.673,A -85,B 0,C 180,E1 -4763.833,E2 -4763.833} C_VEL
LIN {X 0,Y 523.384,Z 779.368,A -85,B 0,C 180,E1 -4764.991,E2 -4764.991} C_VEL
LIN {X 0,Y 523.444,Z 782.954,A -85,B 0,C 180,E1 -4766.149,E2 -4766.149} C_VEL
LIN {X 0,Y 523.368,Z 784.804,A -85,B 0,C 180,E1 -4766.92,E2 -4766.92} C_VEL
LIN {X 0,Y 523.335,Z 786.191,A -85,B 0,C 180,E1 -4767.69,E2 -4767.69} C_VEL
LIN {X 0,Y 523.25,Z 787.784,A -85,B 0,C 180,E1 -4769.229,E2 -4769.229} C_VEL
LIN {X 0,Y 523.246,Z 788,A -85,B 0,C 180,E1 -4769.999,E2 -4769.999} C_VEL
LIN {X 0,Y 523.274,Z 787.185,A -85,B 0,C 180,E1 -4771.538,E2 -4771.538} C_VEL
LIN {X 0,Y 523.334,Z 786.197,A -85,B 0,C 180,E1 -4772.308,E2 -4772.308} C_VEL
LIN {X 0,Y 523.367,Z 784.813,A -85,B 0,C 180,E1 -4773.078,E2 -4773.078} C_VEL
LIN {X 0,Y 523.441,Z 781.899,A -85,B 0,C 180,E1 -4774.234,E2 -4774.234} C_VEL
LIN {X 0,Y 523.464,Z 777.953,A -85,B 0,C 180,E1 -4775.391,E2 -4775.391} C_VEL
LIN {X 0,Y 523.518,Z 772.752,A -85,B 0,C 180,E1 -4776.576,E2 -4776.576} C_VEL
LIN {X 0,Y 523.664,Z 766.473,A -85,B 0,C 180,E1 -4777.711,E2 -4777.711} C_VEL
LIN {X 0,Y 523.851,Z 758.422,A -85,B 0,C 180,E1 -4778.874,E2 -4778.874} C_VEL
LIN {X 0,Y 524.08,Z 750.126,A -85,B 0,C 180,E1 -4779.843,E2 -4779.843} C_VEL
LIN {X 0,Y 524.317,Z 739.987,A -85,B 0,C 180,E1 -4780.815,E2 -4780.815} C_VEL
LIN {X 0,Y 524.642,Z 728.478,A -85,B 0,C 180,E1 -4781.694,E2 -4781.694} C_VEL
LIN {X 0,Y 524.878,Z 717.403,A -85,B 0,C 180,E1 -4782.369,E2 -4782.369} C_VEL
LIN {X 0,Y 525.126,Z 705.059,A -85,B 0,C 180,E1 -4782.953,E2 -4782.953} C_VEL
LIN {X 0,Y 525.355,Z 692.142,A -85,B 0,C 180,E1 -4783.39,E2 -4783.39} C_VEL
LIN {X 0,Y 525.563,Z 678.501,A -85,B 0,C 180,E1 -4783.68,E2 -4783.68} C_VEL
LIN {X 0,Y 525.823,Z 581.914,A -85,B 0,C 180,E1 -4785.006,E2 -4785.006} C_VEL
LIN {X 0,Y 524.633,Z 572.362,A -85,B 0,C 180,E1 -4785.19,E2 -4785.19} C_VEL
LIN {X 0,Y 525.098,Z 545.564,A -85,B 0,C 180,E1 -4788.256,E2 -4788.256} C_VEL
LIN {X 0,Y 525.619,Z 518.709,A -85,B 0,C 180,E1 -4791.366,E2 -4791.366} C_VEL
LIN {X 0,Y 526.197,Z 494.205,A -85,B 0,C 180,E1 -4794.247,E2 -4794.247} C_VEL
LIN {X 0,Y 526.653,Z 472.494,A -85,B 0,C 180,E1 -4796.855,E2 -4796.855} C_VEL
LIN {X 0,Y 525.049,Z 464.223,A -85,B 0,C 180,E1 -4797.94,E2 -4797.94} C_VEL
LIN {X 0,Y 523.977,Z 459.346,A -85,B 0,C 180,E1 -4798.624,E2 -4798.624} C_VEL
LIN {X 0,Y 523.913,Z 459.225,A -85,B 0,C 180,E1 -4801.543,E2 -4801.543} C_VEL
LIN {X 0,Y 523.911,Z 459.227,A -85,B 0,C 180,E1 -4804.29,E2 -4804.29} C_VEL
LIN {X 0,Y 523.875,Z 459.223,A -85,B 0,C 180,E1 -4807.133,E2 -4807.133} C_VEL
LIN {X 0,Y 523.905,Z 459.228,A -85,B 0,C 180,E1 -4810.125,E2 -4810.125} C_VEL
LIN {X 0,Y 523.881,Z 459.222,A -85,B 0,C 180,E1 -4813.169,E2 -4813.169} C_VEL
LIN {X 0,Y 523.919,Z 459.221,A -85,B 0,C 180,E1 -4815.769,E2 -4815.769} C_VEL
LIN {X 0,Y 523.908,Z 459.22,A -85,B 0,C 180,E1 -4818.904,E2 -4818.904} C_VEL
LIN {X 0,Y 523.902,Z 459.224,A -85,B 0,C 180,E1 -4821.897,E2 -4821.897} C_VEL
LIN {X 0,Y 523.912,Z 459.22,A -85,B 0,C 180,E1 -4824.91,E2 -4824.91} C_VEL
LIN {X 0,Y 523.924,Z 459.218,A -85,B 0,C 180,E1 -4827.679,E2 -4827.679} C_VEL
LIN {X 0,Y 523.941,Z 459.219,A -85,B 0,C 180,E1 -4830.676,E2 -4830.676} C_VEL
LIN {X 0,Y 523.932,Z 459.218,A -85,B 0,C 180,E1 -4832.866,E2 -4832.866} C_VEL
LIN {X 0,Y 523.922,Z 459.219,A -85,B 0,C 180,E1 -4835.802,E2 -4835.802} C_VEL
LIN {X 0,Y 523.932,Z 459.22,A -85,B 0,C 180,E1 -4838.766,E2 -4838.766} C_VEL
LIN {X 0,Y 523.927,Z 459.217,A -85,B 0,C 180,E1 -4841.22,E2 -4841.22} C_VEL
LIN {X 0,Y 523.916,Z 459.218,A -85,B 0,C 180,E1 -4843.638,E2 -4843.638} C_VEL
LIN {X 0,Y 523.918,Z 459.221,A -85,B 0,C 180,E1 -4846.027,E2 -4846.027} C_VEL
LIN {X 0,Y 523.999,Z 459.216,A -85,B 0,C 180,E1 -4848.394,E2 -4848.394} C_VEL
LIN {X 0,Y 523.985,Z 459.209,A -85,B 0,C 180,E1 -4851.515,E2 -4851.515} C_VEL
LIN {X 0,Y 524.062,Z 459.208,A -85,B 0,C 180,E1 -4854.613,E2 -4854.613} C_VEL
LIN {X 0,Y 524.093,Z 459.196,A -85,B 0,C 180,E1 -4857.694,E2 -4857.694} C_VEL
LIN {X 0,Y 524.113,Z 459.2,A -85,B 0,C 180,E1 -4860.768,E2 -4860.768} C_VEL
LIN {X 0,Y 524.06,Z 459.202,A -85,B 0,C 180,E1 -4863.075,E2 -4863.075} C_VEL
LIN {X 0,Y 524.021,Z 459.208,A -85,B 0,C 180,E1 -4866.159,E2 -4866.159} C_VEL
LIN {X 0,Y 523.994,Z 459.216,A -85,B 0,C 180,E1 -4868.484,E2 -4868.484} C_VEL
LIN {X 0,Y 523.994,Z 459.208,A -85,B 0,C 180,E1 -4871.743,E2 -4871.743} C_VEL
LIN {X 0,Y 523.979,Z 459.214,A -85,B 0,C 180,E1 -4875.053,E2 -4875.053} C_VEL
LIN {X 0,Y 523.95,Z 459.215,A -85,B 0,C 180,E1 -4877.969,E2 -4877.969} C_VEL
LIN {X 0,Y 523.959,Z 459.218,A -85,B 0,C 180,E1 -4880.41,E2 -4880.41} C_VEL
LIN {X 0,Y 523.903,Z 459.226,A -85,B 0,C 180,E1 -4882.894,E2 -4882.894} C_VEL
LIN {X 0,Y 523.939,Z 459.216,A -85,B 0,C 180,E1 -4885.419,E2 -4885.419} C_VEL
LIN {X 0,Y 523.957,Z 459.214,A -85,B 0,C 180,E1 -4887.999,E2 -4887.999} C_VEL
LIN {X 0,Y 523.934,Z 459.224,A -85,B 0,C 180,E1 -4890.856,E2 -4890.856} C_VEL
LIN {X 0,Y 523.95,Z 459.214,A -85,B 0,C 180,E1 -4893.736,E2 -4893.736} C_VEL
LIN {X 0,Y 523.909,Z 459.222,A -85,B 0,C 180,E1 -4896.405,E2 -4896.405} C_VEL
LIN {X 0,Y 523.912,Z 459.224,A -85,B 0,C 180,E1 -4899.085,E2 -4899.085} C_VEL
LIN {X 0,Y 523.946,Z 459.215,A -85,B 0,C 180,E1 -4902.119,E2 -4902.119} C_VEL
LIN {X 0,Y 523.945,Z 459.218,A -85,B 0,C 180,E1 -4905.31,E2 -4905.31} C_VEL
LIN {X 0,Y 523.914,Z 459.226,A -85,B 0,C 180,E1 -4906.93,E2 -4906.93} C_VEL
LIN {X 0,Y 523.251,Z 459.303,A -85,B 0,C 180,E1 -4907.572,E2 -4907.572} C_VEL
LIN {X 0,Y 520.415,Z 459.659,A -85,B 0,C 180,E1 -4908.613,E2 -4908.613} C_VEL
LIN {X 0,Y 518.016,Z 459.955,A -85,B 0,C 180,E1 -4909.453,E2 -4909.453} C_VEL
LIN {X 0,Y 516.985,Z 460.082,A -85,B 0,C 180,E1 -4910.101,E2 -4910.101} C_VEL
LIN {X 0,Y 516.901,Z 460.094,A -85,B 0,C 180,E1 -4910.32,E2 -4910.32} C_VEL
LIN {X 0,Y 516.874,Z 460.099,A -85,B 0,C 180,E1 -4913.343,E2 -4913.343} C_VEL
LIN {X 0,Y 516.902,Z 460.092,A -85,B 0,C 180,E1 -4916.122,E2 -4916.122} C_VEL
LIN {X 0,Y 516.884,Z 460.103,A -85,B 0,C 180,E1 -4918.937,E2 -4918.937} C_VEL
LIN {X 0,Y 516.913,Z 460.092,A -85,B 0,C 180,E1 -4921.586,E2 -4921.586} C_VEL
LIN {X 0,Y 516.925,Z 460.089,A -85,B 0,C 180,E1 -4924.212,E2 -4924.212} C_VEL
LIN {X 0,Y 516.866,Z 460.102,A -85,B 0,C 180,E1 -4926.778,E2 -4926.778} C_VEL
LIN {X 0,Y 516.934,Z 460.089,A -85,B 0,C 180,E1 -4929.733,E2 -4929.733} C_VEL
LIN {X 0,Y 516.925,Z 460.092,A -85,B 0,C 180,E1 -4932.598,E2 -4932.598} C_VEL
LIN {X 0,Y 516.938,Z 460.096,A -85,B 0,C 180,E1 -4935.031,E2 -4935.031} C_VEL
LIN {X 0,Y 516.962,Z 460.084,A -85,B 0,C 180,E1 -4938.235,E2 -4938.235} C_VEL
LIN {X 0,Y 516.967,Z 460.091,A -85,B 0,C 180,E1 -4941.401,E2 -4941.401} C_VEL
LIN {X 0,Y 517.013,Z 460.083,A -85,B 0,C 180,E1 -4943.758,E2 -4943.758} C_VEL
LIN {X 0,Y 517.084,Z 460.078,A -85,B 0,C 180,E1 -4947.664,E2 -4947.664} C_VEL
LIN {X 0,Y 517.04,Z 460.234,A -85,B 0,C 180,E1 -4948.93,E2 -4948.93} C_VEL
LIN {X 0,Y 517.277,Z 461.212,A -85,B 0,C 180,E1 -4949.065,E2 -4949.065} C_VEL
LIN {X 0,Y 519.212,Z 467.481,A -85,B 0,C 180,E1 -4949.226,E2 -4949.226} C_VEL
LIN {X 0,Y 518.86,Z 540.897,A -85,B 0,C 180,E1 -4950.268,E2 -4950.268} C_VEL
LIN {X 0,Y 518.781,Z 553.809,A -85,B 0,C 180,E1 -4950.608,E2 -4950.608} C_VEL
LIN {X 0,Y 518.613,Z 565.736,A -85,B 0,C 180,E1 -4951.069,E2 -4951.069} C_VEL
LIN {X 0,Y 518.462,Z 576.965,A -85,B 0,C 180,E1 -4951.652,E2 -4951.652} C_VEL
LIN {X 0,Y 518.196,Z 588.548,A -85,B 0,C 180,E1 -4952.43,E2 -4952.43} C_VEL
LIN {X 0,Y 517.847,Z 598.939,A -85,B 0,C 180,E1 -4953.308,E2 -4953.308} C_VEL
LIN {X 0,Y 517.611,Z 608.278,A -85,B 0,C 180,E1 -4954.284,E2 -4954.284} C_VEL
LIN {X 0,Y 517.337,Z 615.971,A -85,B 0,C 180,E1 -4955.263,E2 -4955.263} C_VEL
LIN {X 0,Y 517.193,Z 623.457,A -85,B 0,C 180,E1 -4956.438,E2 -4956.438} C_VEL
LIN {X 0,Y 516.954,Z 630.398,A -85,B 0,C 180,E1 -4957.815,E2 -4957.815} C_VEL
LIN {X 0,Y 516.791,Z 635.024,A -85,B 0,C 180,E1 -4958.999,E2 -4958.999} C_VEL
LIN {X 0,Y 516.691,Z 638.554,A -85,B 0,C 180,E1 -4960.186,E2 -4960.186} C_VEL
LIN {X 0,Y 516.631,Z 641.511,A -85,B 0,C 180,E1 -4961.636,E2 -4961.636} C_VEL
LIN {X 0,Y 516.596,Z 642.668,A -85,B 0,C 180,E1 -4962.573,E2 -4962.573} C_VEL
LIN {X 0,Y 516.546,Z 643.246,A -85,B 0,C 180,E1 -4963.375,E2 -4963.375} C_VEL
LIN {X 0,Y 516.525,Z 643.379,A -85,B 0,C 180,E1 -4964.178,E2 -4964.178} C_VEL
LIN {X 0,Y 516.567,Z 643.097,A -85,B 0,C 180,E1 -4964.991,E2 -4964.991} C_VEL
LIN {X 0,Y 516.573,Z 642.434,A -85,B 0,C 180,E1 -4965.791,E2 -4965.791} C_VEL
LIN {X 0,Y 516.608,Z 641.339,A -85,B 0,C 180,E1 -4966.601,E2 -4966.601} C_VEL
LIN {X 0,Y 516.716,Z 638.881,A -85,B 0,C 180,E1 -4967.808,E2 -4967.808} C_VEL
LIN {X 0,Y 516.807,Z 635.275,A -85,B 0,C 180,E1 -4969.05,E2 -4969.05} C_VEL
LIN {X 0,Y 516.983,Z 630.496,A -85,B 0,C 180,E1 -4970.282,E2 -4970.282} C_VEL
LIN {X 0,Y 517.163,Z 624.316,A -85,B 0,C 180,E1 -4971.527,E2 -4971.527} C_VEL
LIN {X 0,Y 517.422,Z 616.372,A -85,B 0,C 180,E1 -4972.795,E2 -4972.795} C_VEL
LIN {X 0,Y 517.634,Z 608.317,A -85,B 0,C 180,E1 -4973.825,E2 -4973.825} C_VEL
LIN {X 0,Y 517.911,Z 598.14,A -85,B 0,C 180,E1 -4974.878,E2 -4974.878} C_VEL
LIN {X 0,Y 518.208,Z 588.002,A -85,B 0,C 180,E1 -4975.722,E2 -4975.722} C_VEL
LIN {X 0,Y 518.505,Z 576.194,A -85,B 0,C 180,E1 -4976.496,E2 -4976.496} C_VEL
LIN {X 0,Y 518.662,Z 564.102,A -85,B 0,C 180,E1 -4977.106,E2 -4977.106} C_VEL
LIN {X 0,Y 518.821,Z 551.691,A -85,B 0,C 180,E1 -4977.562,E2 -4977.562} C_VEL
LIN {X 0,Y 518.867,Z 539.157,A -85,B 0,C 180,E1 -4977.86,E2 -4977.86} C_VEL
LIN {X 0,Y 519.131,Z 466.969,A -85,B 0,C 180,E1 -4978.882,E2 -4978.882} C_VEL
LIN {X 0,Y 517.084,Z 460.979,A -85,B 0,C 180,E1 -4979.06,E2 -4979.06} C_VEL
LIN {X 0,Y 516.947,Z 460.157,A -85,B 0,C 180,E1 -4979.22,E2 -4979.22} C_VEL
LIN {X 0,Y 516.897,Z 460.1,A -85,B 0,C 180,E1 -4982.544,E2 -4982.544} C_VEL
LIN {X 0,Y 516.869,Z 460.102,A -85,B 0,C 180,E1 -4985.33,E2 -4985.33} C_VEL
LIN {X 0,Y 516.883,Z 460.096,A -85,B 0,C 180,E1 -4987.944,E2 -4987.944} C_VEL
LIN {X 0,Y 516.887,Z 460.101,A -85,B 0,C 180,E1 -4990.743,E2 -4990.743} C_VEL
LIN {X 0,Y 516.886,Z 460.099,A -85,B 0,C 180,E1 -4992.832,E2 -4992.832} C_VEL
LIN {X 0,Y 516.899,Z 460.101,A -85,B 0,C 180,E1 -4995.008,E2 -4995.008} C_VEL
LIN {X 0,Y 516.918,Z 460.096,A -85,B 0,C 180,E1 -4998.4,E2 -4998.4} C_VEL
LIN {X 0,Y 516.884,Z 460.099,A -85,B 0,C 180,E1 -5001.285,E2 -5001.285} C_VEL
LIN {X 0,Y 516.929,Z 460.308,A -85,B 0,C 180,E1 -5002.805,E2 -5002.805} C_VEL
LIN {X 0,Y 518.436,Z 468.137,A -85,B 0,C 180,E1 -5004.105,E2 -5004.105} C_VEL
LIN {X 0,Y 518.264,Z 480.398,A -85,B 0,C 180,E1 -5006.013,E2 -5006.013} C_VEL
LIN {X 0,Y 517.941,Z 496.052,A -85,B 0,C 180,E1 -5008.45,E2 -5008.45} C_VEL
LIN {X 0,Y 517.516,Z 515.001,A -85,B 0,C 180,E1 -5011.4,E2 -5011.4} C_VEL
LIN {X 0,Y 517.531,Z 517.182,A -85,B 0,C 180,E1 -5011.683,E2 -5011.683} C_VEL
LIN {X 0,Y 519.114,Z 526.852,A -85,B 0,C 180,E1 -5011.889,E2 -5011.889} C_VEL
LIN {X 0,Y 518.588,Z 625.138,A -85,B 0,C 180,E1 -5013.299,E2 -5013.299} C_VEL
LIN {X 0,Y 518.379,Z 638.376,A -85,B 0,C 180,E1 -5013.64,E2 -5013.64} C_VEL
LIN {X 0,Y 518.108,Z 650.441,A -85,B 0,C 180,E1 -5014.112,E2 -5014.112} C_VEL
LIN {X 0,Y 517.904,Z 661.654,A -85,B 0,C 180,E1 -5014.694,E2 -5014.694} C_VEL
LIN {X 0,Y 517.591,Z 673.351,A -85,B 0,C 180,E1 -5015.472,E2 -5015.472} C_VEL
LIN {X 0,Y 517.237,Z 683.93,A -85,B 0,C 180,E1 -5016.37,E2 -5016.37} C_VEL
LIN {X 0,Y 517.024,Z 692.462,A -85,B 0,C 180,E1 -5017.249,E2 -5017.249} C_VEL
LIN {X 0,Y 516.75,Z 701.933,A -85,B 0,C 180,E1 -5018.457,E2 -5018.457} C_VEL
LIN {X 0,Y 516.545,Z 709.212,A -85,B 0,C 180,E1 -5019.618,E2 -5019.618} C_VEL
LIN {X 0,Y 516.428,Z 715.818,A -85,B 0,C 180,E1 -5020.937,E2 -5020.937} C_VEL
LIN {X 0,Y 516.372,Z 719.099,A -85,B 0,C 180,E1 -5021.758,E2 -5021.758} C_VEL
LIN {X 0,Y 516.276,Z 723.002,A -85,B 0,C 180,E1 -5022.982,E2 -5022.982} C_VEL
LIN {X 0,Y 516.194,Z 725.768,A -85,B 0,C 180,E1 -5024.199,E2 -5024.199} C_VEL
LIN {X 0,Y 516.187,Z 727.273,A -85,B 0,C 180,E1 -5025.171,E2 -5025.171} C_VEL
LIN {X 0,Y 516.174,Z 728.33,A -85,B 0,C 180,E1 -5026.617,E2 -5026.617} C_VEL
LIN {X 0,Y 516.232,Z 727.991,A -85,B 0,C 180,E1 -5028.217,E2 -5028.217} C_VEL
LIN {X 0,Y 516.282,Z 727.181,A -85,B 0,C 180,E1 -5029.014,E2 -5029.014} C_VEL
LIN {X 0,Y 516.234,Z 724.287,A -85,B 0,C 180,E1 -5030.598,E2 -5030.598} C_VEL
LIN {X 0,Y 516.333,Z 720.984,A -85,B 0,C 180,E1 -5031.783,E2 -5031.783} C_VEL
LIN {X 0,Y 516.429,Z 716.643,A -85,B 0,C 180,E1 -5032.965,E2 -5032.965} C_VEL
LIN {X 0,Y 516.561,Z 710.022,A -85,B 0,C 180,E1 -5034.339,E2 -5034.339} C_VEL
LIN {X 0,Y 516.665,Z 704.117,A -85,B 0,C 180,E1 -5035.319,E2 -5035.319} C_VEL
LIN {X 0,Y 516.835,Z 697.073,A -85,B 0,C 180,E1 -5036.297,E2 -5036.297} C_VEL
LIN {X 0,Y 517.122,Z 688.57,A -85,B 0,C 180,E1 -5037.274,E2 -5037.274} C_VEL
LIN {X 0,Y 517.429,Z 678.054,A -85,B 0,C 180,E1 -5038.249,E2 -5038.249} C_VEL
LIN {X 0,Y 517.712,Z 667.616,A -85,B 0,C 180,E1 -5039.028,E2 -5039.028} C_VEL
LIN {X 0,Y 517.964,Z 656.1,A -85,B 0,C 180,E1 -5039.709,E2 -5039.709} C_VEL
LIN {X 0,Y 518.315,Z 644.067,A -85,B 0,C 180,E1 -5040.243,E2 -5040.243} C_VEL
LIN {X 0,Y 518.467,Z 631.99,A -85,B 0,C 180,E1 -5040.631,E2 -5040.631} C_VEL
LIN {X 0,Y 518.622,Z 618.52,A -85,B 0,C 180,E1 -5040.898,E2 -5040.898} C_VEL
LIN {X 0,Y 519.06,Z 526.574,A -85,B 0,C 180,E1 -5042.207,E2 -5042.207} C_VEL
LIN {X 0,Y 517.635,Z 517.482,A -85,B 0,C 180,E1 -5042.408,E2 -5042.408} C_VEL
LIN {X 0,Y 517.868,Z 498.855,A -85,B 0,C 180,E1 -5045.256,E2 -5045.256} C_VEL
LIN {X 0,Y 518.163,Z 483.614,A -85,B 0,C 180,E1 -5047.578,E2 -5047.578} C_VEL
LIN {X 0,Y 518.32,Z 467.837,A -85,B 0,C 180,E1 -5049.956,E2 -5049.956} C_VEL
LIN {X 0,Y 516.987,Z 460.171,A -85,B 0,C 180,E1 -5051.187,E2 -5051.187} C_VEL
LIN {X 0,Y 516.876,Z 460.1,A -85,B 0,C 180,E1 -5054.167,E2 -5054.167} C_VEL
LIN {X 0,Y 516.895,Z 460.098,A -85,B 0,C 180,E1 -5056.591,E2 -5056.591} C_VEL
LIN {X 0,Y 516.898,Z 460.102,A -85,B 0,C 180,E1 -5059.046,E2 -5059.046} C_VEL
LIN {X 0,Y 516.892,Z 460.098,A -85,B 0,C 180,E1 -5061.538,E2 -5061.538} C_VEL
LIN {X 0,Y 516.885,Z 460.098,A -85,B 0,C 180,E1 -5064.356,E2 -5064.356} C_VEL
LIN {X 0,Y 516.932,Z 460.091,A -85,B 0,C 180,E1 -5067.533,E2 -5067.533} C_VEL
LIN {X 0,Y 516.895,Z 460.096,A -85,B 0,C 180,E1 -5070.204,E2 -5070.204} C_VEL
LIN {X 0,Y 516.903,Z 460.099,A -85,B 0,C 180,E1 -5072.947,E2 -5072.947} C_VEL
LIN {X 0,Y 516.879,Z 460.096,A -85,B 0,C 180,E1 -5075.78,E2 -5075.78} C_VEL
LIN {X 0,Y 516.888,Z 460.103,A -85,B 0,C 180,E1 -5078.716,E2 -5078.716} C_VEL
LIN {X 0,Y 516.92,Z 460.092,A -85,B 0,C 180,E1 -5081.775,E2 -5081.775} C_VEL
LIN {X 0,Y 516.903,Z 460.096,A -85,B 0,C 180,E1 -5085.006,E2 -5085.006} C_VEL
LIN {X 0,Y 516.921,Z 460.097,A -85,B 0,C 180,E1 -5088.398,E2 -5088.398} C_VEL
LIN {X 0,Y 516.884,Z 460.089,A -85,B 0,C 180,E1 -5091.283,E2 -5091.283} C_VEL
LIN {X 0,Y 516.873,Z 460.104,A -85,B 0,C 180,E1 -5094.219,E2 -5094.219} C_VEL
LIN {X 0,Y 516.888,Z 460.098,A -85,B 0,C 180,E1 -5097.051,E2 -5097.051} C_VEL
LIN {X 0,Y 516.893,Z 460.101,A -85,B 0,C 180,E1 -5099.795,E2 -5099.795} C_VEL
LIN {X 0,Y 516.943,Z 460.326,A -85,B 0,C 180,E1 -5101.28,E2 -5101.28} C_VEL
LIN {X 0,Y 519.578,Z 472.617,A -85,B 0,C 180,E1 -5102.963,E2 -5102.963} C_VEL
LIN {X 0,Y 519.326,Z 488.594,A -85,B 0,C 180,E1 -5104.912,E2 -5104.912} C_VEL
LIN {X 0,Y 518.757,Z 513.735,A -85,B 0,C 180,E1 -5107.916,E2 -5107.916} C_VEL
LIN {X 0,Y 518.174,Z 540.067,A -85,B 0,C 180,E1 -5111.002,E2 -5111.002} C_VEL
LIN {X 0,Y 517.621,Z 567.986,A -85,B 0,C 180,E1 -5114.242,E2 -5114.242} C_VEL
LIN {X 0,Y 517.591,Z 571.344,A -85,B 0,C 180,E1 -5114.605,E2 -5114.605} C_VEL
LIN {X 0,Y 519.052,Z 584.527,A -85,B 0,C 180,E1 -5114.845,E2 -5114.845} C_VEL
LIN {X 0,Y 518.634,Z 681.635,A -85,B 0,C 180,E1 -5116.206,E2 -5116.206} C_VEL
LIN {X 0,Y 518.351,Z 695.046,A -85,B 0,C 180,E1 -5116.548,E2 -5116.548} C_VEL
LIN {X 0,Y 518.084,Z 708.489,A -85,B 0,C 180,E1 -5117.065,E2 -5117.065} C_VEL
LIN {X 0,Y 517.772,Z 720.646,A -85,B 0,C 180,E1 -5117.707,E2 -5117.707} C_VEL
LIN {X 0,Y 517.448,Z 732.879,A -85,B 0,C 180,E1 -5118.542,E2 -5118.542} C_VEL
LIN {X 0,Y 517.163,Z 743.256,A -85,B 0,C 180,E1 -5119.427,E2 -5119.427} C_VEL
LIN {X 0,Y 516.927,Z 752.61,A -85,B 0,C 180,E1 -5120.412,E2 -5120.412} C_VEL
LIN {X 0,Y 516.686,Z 761.734,A -85,B 0,C 180,E1 -5121.591,E2 -5121.591} C_VEL
LIN {X 0,Y 516.512,Z 769.093,A -85,B 0,C 180,E1 -5122.768,E2 -5122.768} C_VEL
LIN {X 0,Y 516.455,Z 775.824,A -85,B 0,C 180,E1 -5124.141,E2 -5124.141} C_VEL
LIN {X 0,Y 516.272,Z 780.256,A -85,B 0,C 180,E1 -5125.314,E2 -5125.314} C_VEL
LIN {X 0,Y 516.373,Z 782.63,A -85,B 0,C 180,E1 -5126.097,E2 -5126.097} C_VEL
LIN {X 0,Y 516.283,Z 784.531,A -85,B 0,C 180,E1 -5126.877,E2 -5126.877} C_VEL
LIN {X 0,Y 516.261,Z 785.965,A -85,B 0,C 180,E1 -5127.658,E2 -5127.658} C_VEL
LIN {X 0,Y 516.16,Z 787.597,A -85,B 0,C 180,E1 -5129.219,E2 -5129.219} C_VEL
LIN {X 0,Y 516.154,Z 787.819,A -85,B 0,C 180,E1 -5129.999,E2 -5129.999} C_VEL
LIN {X 0,Y 516.16,Z 787.599,A -85,B 0,C 180,E1 -5130.779,E2 -5130.779} C_VEL
LIN {X 0,Y 516.261,Z 785.972,A -85,B 0,C 180,E1 -5132.339,E2 -5132.339} C_VEL
LIN {X 0,Y 516.282,Z 784.541,A -85,B 0,C 180,E1 -5133.12,E2 -5133.12} C_VEL
LIN {X 0,Y 516.326,Z 781.533,A -85,B 0,C 180,E1 -5134.292,E2 -5134.292} C_VEL
LIN {X 0,Y 516.405,Z 777.468,A -85,B 0,C 180,E1 -5135.465,E2 -5135.465} C_VEL
LIN {X 0,Y 516.462,Z 772.056,A -85,B 0,C 180,E1 -5136.676,E2 -5136.676} C_VEL
LIN {X 0,Y 516.577,Z 765.651,A -85,B 0,C 180,E1 -5137.818,E2 -5137.818} C_VEL
LIN {X 0,Y 516.787,Z 757.46,A -85,B 0,C 180,E1 -5138.996,E2 -5138.996} C_VEL
LIN {X 0,Y 517.021,Z 749.133,A -85,B 0,C 180,E1 -5139.979,E2 -5139.979} C_VEL
LIN {X 0,Y 517.276,Z 738.993,A -85,B 0,C 180,E1 -5140.964,E2 -5140.964} C_VEL
LIN {X 0,Y 517.621,Z 727.662,A -85,B 0,C 180,E1 -5141.843,E2 -5141.843} C_VEL
LIN {X 0,Y 517.897,Z 716.407,A -85,B 0,C 180,E1 -5142.539,E2 -5142.539} C_VEL
LIN {X 0,Y 518.197,Z 704.066,A -85,B 0,C 180,E1 -5143.129,E2 -5143.129} C_VEL
LIN {X 0,Y 518.405,Z 691.133,A -85,B 0,C 180,E1 -5143.573,E2 -5143.573} C_VEL
LIN {X 0,Y 518.649,Z 677.48,A -85,B 0,C 180,E1 -5143.866,E2 -5143.866} C_VEL
LIN {X 0,Y 518.988,Z 583.06,A -85,B 0,C 180,E1 -5145.179,E2 -5145.179} C_VEL
LIN {X 0,Y 517.576,Z 571.398,A -85,B 0,C 180,E1 -5145.401,E2 -5145.401} C_VEL
LIN {X 0,Y 518.063,Z 545.848,A -85,B 0,C 180,E1 -5148.363,E2 -5148.363} C_VEL
LIN {X 0,Y 518.62,Z 519.503,A -85,B 0,C 180,E1 -5151.461,E2 -5151.461} C_VEL
LIN {X 0,Y 519.266,Z 495.102,A -85,B 0,C 180,E1 -5154.379,E2 -5154.379} C_VEL
LIN {X 0,Y 519.751,Z 473.303,A -85,B 0,C 180,E1 -5157.037,E2 -5157.037} C_VEL
LIN {X 0,Y 516.937,Z 460.223,A -85,B 0,C 180,E1 -5158.828,E2 -5158.828} C_VEL
LIN {X 0,Y 516.867,Z 460.106,A -85,B 0,C 180,E1 -5162.023,E2 -5162.023} C_VEL
LIN {X 0,Y 516.869,Z 460.099,A -85,B 0,C 180,E1 -5164.824,E2 -5164.824} C_VEL
LIN {X 0,Y 516.856,Z 460.103,A -85,B 0,C 180,E1 -5167.939,E2 -5167.939} C_VEL
LIN {X 0,Y 516.845,Z 460.101,A -85,B 0,C 180,E1 -5170.743,E2 -5170.743} C_VEL
LIN {X 0,Y 516.872,Z 460.1,A -85,B 0,C 180,E1 -5173.902,E2 -5173.902} C_VEL
LIN {X 0,Y 516.872,Z 460.103,A -85,B 0,C 180,E1 -5176.106,E2 -5176.106} C_VEL
LIN {X 0,Y 516.893,Z 460.1,A -85,B 0,C 180,E1 -5178.399,E2 -5178.399} C_VEL
LIN {X 0,Y 516.866,Z 460.096,A -85,B 0,C 180,E1 -5181.282,E2 -5181.282} C_VEL
LIN {X 0,Y 516.856,Z 460.106,A -85,B 0,C 180,E1 -5184.218,E2 -5184.218} C_VEL
LIN {X 0,Y 516.883,Z 460.095,A -85,B 0,C 180,E1 -5187.052,E2 -5187.052} C_VEL
LIN {X 0,Y 516.875,Z 460.097,A -85,B 0,C 180,E1 -5189.795,E2 -5189.795} C_VEL
LIN {X 0,Y 516.909,Z 460.099,A -85,B 0,C 180,E1 -5192.466,E2 -5192.466} C_VEL
LIN {X 0,Y 516.845,Z 460.1,A -85,B 0,C 180,E1 -5195.068,E2 -5195.068} C_VEL
LIN {X 0,Y 516.856,Z 460.098,A -85,B 0,C 180,E1 -5197.621,E2 -5197.621} C_VEL
LIN {X 0,Y 516.916,Z 460.095,A -85,B 0,C 180,E1 -5200.129,E2 -5200.129} C_VEL
LIN {X 0,Y 516.905,Z 460.098,A -85,B 0,C 180,E1 -5202.595,E2 -5202.595} C_VEL
LIN {X 0,Y 516.926,Z 460.09,A -85,B 0,C 180,E1 -5205.029,E2 -5205.029} C_VEL
LIN {X 0,Y 516.952,Z 460.091,A -85,B 0,C 180,E1 -5208.233,E2 -5208.233} C_VEL
LIN {X 0,Y 516.951,Z 460.086,A -85,B 0,C 180,E1 -5211.399,E2 -5211.399} C_VEL
LIN {X 0,Y 516.983,Z 460.082,A -85,B 0,C 180,E1 -5213.756,E2 -5213.756} C_VEL
LIN {X 0,Y 517,Z 460.084,A -85,B 0,C 180,E1 -5216.883,E2 -5216.883} C_VEL
LIN {X 0,Y 517.066,Z 460.073,A -85,B 0,C 180,E1 -5220,E2 -5220} C_VEL
LIN {X 0,Y 517.001,Z 460.082,A -85,B 0,C 180,E1 -5223.117,E2 -5223.117} C_VEL
LIN {X 0,Y 516.987,Z 460.085,A -85,B 0,C 180,E1 -5226.243,E2 -5226.243} C_VEL
LIN {X 0,Y 516.943,Z 460.087,A -85,B 0,C 180,E1 -5229.389,E2 -5229.389} C_VEL
LIN {X 0,Y 516.943,Z 460.087,A -85,B 0,C 180,E1 -5231.81,E2 -5231.81} C_VEL
LIN {X 0,Y 516.932,Z 460.091,A -85,B 0,C 180,E1 -5235.148,E2 -5235.148} C_VEL
LIN {X 0,Y 516.911,Z 460.094,A -85,B 0,C 180,E1 -5238.222,E2 -5238.222} C_VEL
LIN {X 0,Y 516.899,Z 460.102,A -85,B 0,C 180,E1 -5240.702,E2 -5240.702} C_VEL
LIN {X 0,Y 516.897,Z 460.094,A -85,B 0,C 180,E1 -5244.072,E2 -5244.072} C_VEL
LIN {X 0,Y 516.913,Z 460.099,A -85,B 0,C 180,E1 -5246.658,E2 -5246.658} C_VEL
LIN {X 0,Y 516.898,Z 460.093,A -85,B 0,C 180,E1 -5249.525,E2 -5249.525} C_VEL
LIN {X 0,Y 516.888,Z 460.099,A -85,B 0,C 180,E1 -5252.545,E2 -5252.545} C_VEL
LIN {X 0,Y 516.87,Z 460.098,A -85,B 0,C 180,E1 -5255.333,E2 -5255.333} C_VEL
LIN {X 0,Y 516.869,Z 460.096,A -85,B 0,C 180,E1 -5257.944,E2 -5257.944} C_VEL
LIN {X 0,Y 516.874,Z 460.103,A -85,B 0,C 180,E1 -5260.742,E2 -5260.742} C_VEL
LIN {X 0,Y 516.893,Z 460.102,A -85,B 0,C 180,E1 -5262.83,E2 -5262.83} C_VEL
LIN {X 0,Y 516.911,Z 460.098,A -85,B 0,C 180,E1 -5265.011,E2 -5265.011} C_VEL
LIN {X 0,Y 516.919,Z 460.092,A -85,B 0,C 180,E1 -5268.398,E2 -5268.398} C_VEL
LIN {X 0,Y 516.901,Z 460.094,A -85,B 0,C 180,E1 -5270.32,E2 -5270.32} C_VEL
LIN {X 0,Y 516.232,Z 460.184,A -85,B 0,C 180,E1 -5270.97,E2 -5270.97} C_VEL
LIN {X 0,Y 513.374,Z 460.538,A -85,B 0,C 180,E1 -5272.025,E2 -5272.025} C_VEL
LIN {X 0,Y 510.954,Z 460.841,A -85,B 0,C 180,E1 -5272.875,E2 -5272.875} C_VEL
LIN {X 0,Y 509.908,Z 460.965,A -85,B 0,C 180,E1 -5273.532,E2 -5273.532} C_VEL
LIN {X 0,Y 509.82,Z 460.974,A -85,B 0,C 180,E1 -5273.754,E2 -5273.754} C_VEL
LIN {X 0,Y 509.853,Z 460.973,A -85,B 0,C 180,E1 -5276.541,E2 -5276.541} C_VEL
LIN {X 0,Y 509.838,Z 460.976,A -85,B 0,C 180,E1 -5279.336,E2 -5279.336} C_VEL
LIN {X 0,Y 509.887,Z 460.966,A -85,B 0,C 180,E1 -5282.056,E2 -5282.056} C_VEL
LIN {X 0,Y 509.87,Z 460.972,A -85,B 0,C 180,E1 -5284.705,E2 -5284.705} C_VEL
LIN {X 0,Y 509.85,Z 460.974,A -85,B 0,C 180,E1 -5287.451,E2 -5287.451} C_VEL
LIN {X 0,Y 509.911,Z 460.963,A -85,B 0,C 180,E1 -5289.846,E2 -5289.846} C_VEL
LIN {X 0,Y 509.881,Z 460.975,A -85,B 0,C 180,E1 -5293.176,E2 -5293.176} C_VEL
LIN {X 0,Y 509.86,Z 460.971,A -85,B 0,C 180,E1 -5295.636,E2 -5295.636} C_VEL
LIN {X 0,Y 509.91,Z 460.968,A -85,B 0,C 180,E1 -5298.876,E2 -5298.876} C_VEL
LIN {X 0,Y 509.949,Z 460.96,A -85,B 0,C 180,E1 -5302.08,E2 -5302.08} C_VEL
LIN {X 0,Y 509.984,Z 460.958,A -85,B 0,C 180,E1 -5304.466,E2 -5304.466} C_VEL
LIN {X 0,Y 510.055,Z 460.953,A -85,B 0,C 180,E1 -5307.632,E2 -5307.632} C_VEL
LIN {X 0,Y 509.974,Z 461.092,A -85,B 0,C 180,E1 -5308.712,E2 -5308.712} C_VEL
LIN {X 0,Y 510.178,Z 462.055,A -85,B 0,C 180,E1 -5308.855,E2 -5308.855} C_VEL
LIN {X 0,Y 512.362,Z 468.624,A -85,B 0,C 180,E1 -5309.031,E2 -5309.031} C_VEL
LIN {X 0,Y 512.003,Z 541.422,A -85,B 0,C 180,E1 -5310.075,E2 -5310.075} C_VEL
LIN {X 0,Y 511.917,Z 554.492,A -85,B 0,C 180,E1 -5310.419,E2 -5310.419} C_VEL
LIN {X 0,Y 511.767,Z 567.564,A -85,B 0,C 180,E1 -5310.936,E2 -5310.936} C_VEL
LIN {X 0,Y 511.537,Z 579.396,A -85,B 0,C 180,E1 -5311.576,E2 -5311.576} C_VEL
LIN {X 0,Y 511.262,Z 590.664,A -85,B 0,C 180,E1 -5312.365,E2 -5312.365} C_VEL
LIN {X 0,Y 510.904,Z 600.861,A -85,B 0,C 180,E1 -5313.254,E2 -5313.254} C_VEL
LIN {X 0,Y 510.678,Z 609.177,A -85,B 0,C 180,E1 -5314.145,E2 -5314.145} C_VEL
LIN {X 0,Y 510.413,Z 616.878,A -85,B 0,C 180,E1 -5315.136,E2 -5315.136} C_VEL
LIN {X 0,Y 510.221,Z 624.392,A -85,B 0,C 180,E1 -5316.328,E2 -5316.328} C_VEL
LIN {X 0,Y 510.012,Z 630.272,A -85,B 0,C 180,E1 -5317.484,E2 -5317.484} C_VEL
LIN {X 0,Y 509.828,Z 635.268,A -85,B 0,C 180,E1 -5318.723,E2 -5318.723} C_VEL
LIN {X 0,Y 509.707,Z 638.983,A -85,B 0,C 180,E1 -5319.926,E2 -5319.926} C_VEL
LIN {X 0,Y 509.643,Z 641.683,A -85,B 0,C 180,E1 -5321.133,E2 -5321.133} C_VEL
LIN {X 0,Y 509.596,Z 642.96,A -85,B 0,C 180,E1 -5321.94,E2 -5321.94} C_VEL
LIN {X 0,Y 509.559,Z 643.843,A -85,B 0,C 180,E1 -5322.75,E2 -5322.75} C_VEL
LIN {X 0,Y 509.522,Z 644.284,A -85,B 0,C 180,E1 -5323.563,E2 -5323.563} C_VEL
LIN {X 0,Y 509.556,Z 643.971,A -85,B 0,C 180,E1 -5325.193,E2 -5325.193} C_VEL
LIN {X 0,Y 509.577,Z 643.199,A -85,B 0,C 180,E1 -5326.013,E2 -5326.013} C_VEL
LIN {X 0,Y 509.612,Z 641.971,A -85,B 0,C 180,E1 -5326.836,E2 -5326.836} C_VEL
LIN {X 0,Y 509.715,Z 639.658,A -85,B 0,C 180,E1 -5327.941,E2 -5327.941} C_VEL
LIN {X 0,Y 509.822,Z 635.56,A -85,B 0,C 180,E1 -5329.321,E2 -5329.321} C_VEL
LIN {X 0,Y 510.054,Z 630.213,A -85,B 0,C 180,E1 -5330.655,E2 -5330.655} C_VEL
LIN {X 0,Y 510.244,Z 624.196,A -85,B 0,C 180,E1 -5331.834,E2 -5331.834} C_VEL
LIN {X 0,Y 510.478,Z 617.694,A -85,B 0,C 180,E1 -5332.868,E2 -5332.868} C_VEL
LIN {X 0,Y 510.728,Z 609.386,A -85,B 0,C 180,E1 -5333.951,E2 -5333.951} C_VEL
LIN {X 0,Y 511.011,Z 599.874,A -85,B 0,C 180,E1 -5334.958,E2 -5334.958} C_VEL
LIN {X 0,Y 511.333,Z 589.122,A -85,B 0,C 180,E1 -5335.875,E2 -5335.875} C_VEL
LIN {X 0,Y 511.636,Z 578.015,A -85,B 0,C 180,E1 -5336.622,E2 -5336.622} C_VEL
LIN {X 0,Y 511.824,Z 565.323,A -85,B 0,C 180,E1 -5337.277,E2 -5337.277} C_VEL
LIN {X 0,Y 511.953,Z 552.972,A -85,B 0,C 180,E1 -5337.741,E2 -5337.741} C_VEL
LIN {X 0,Y 512.048,Z 540.581,A -85,B 0,C 180,E1 -5338.044,E2 -5338.044} C_VEL
LIN {X 0,Y 512.358,Z 468.455,A -85,B 0,C 180,E1 -5339.084,E2 -5339.084} C_VEL
LIN {X 0,Y 510.031,Z 461.797,A -85,B 0,C 180,E1 -5339.288,E2 -5339.288} C_VEL
LIN {X 0,Y 509.894,Z 461.022,A -85,B 0,C 180,E1 -5339.466,E2 -5339.466} C_VEL
LIN {X 0,Y 509.87,Z 460.977,A -85,B 0,C 180,E1 -5342.774,E2 -5342.774} C_VEL
LIN {X 0,Y 509.829,Z 460.977,A -85,B 0,C 180,E1 -5345.579,E2 -5345.579} C_VEL
LIN {X 0,Y 509.853,Z 460.974,A -85,B 0,C 180,E1 -5348.339,E2 -5348.339} C_VEL
LIN {X 0,Y 509.859,Z 460.972,A -85,B 0,C 180,E1 -5351.426,E2 -5351.426} C_VEL
LIN {X 0,Y 509.843,Z 460.98,A -85,B 0,C 180,E1 -5354.671,E2 -5354.671} C_VEL
LIN {X 0,Y 509.837,Z 460.976,A -85,B 0,C 180,E1 -5357.511,E2 -5357.511} C_VEL
LIN {X 0,Y 509.85,Z 460.979,A -85,B 0,C 180,E1 -5360.648,E2 -5360.648} C_VEL
LIN {X 0,Y 509.875,Z 461.146,A -85,B 0,C 180,E1 -5362.618,E2 -5362.618} C_VEL
LIN {X 0,Y 511.551,Z 470.336,A -85,B 0,C 180,E1 -5364.154,E2 -5364.154} C_VEL
LIN {X 0,Y 511.245,Z 488.464,A -85,B 0,C 180,E1 -5366.99,E2 -5366.99} C_VEL
LIN {X 0,Y 510.743,Z 508.359,A -85,B 0,C 180,E1 -5370.102,E2 -5370.102} C_VEL
LIN {X 0,Y 510.551,Z 517.19,A -85,B 0,C 180,E1 -5371.454,E2 -5371.454} C_VEL
LIN {X 0,Y 511.884,Z 525.046,A -85,B 0,C 180,E1 -5371.642,E2 -5371.642} C_VEL
LIN {X 0,Y 512.248,Z 529.969,A -85,B 0,C 180,E1 -5371.727,E2 -5371.727} C_VEL
LIN {X 0,Y 511.683,Z 625.796,A -85,B 0,C 180,E1 -5373.131,E2 -5373.131} C_VEL
LIN {X 0,Y 511.455,Z 639.479,A -85,B 0,C 180,E1 -5373.497,E2 -5373.497} C_VEL
LIN {X 0,Y 511.166,Z 650.906,A -85,B 0,C 180,E1 -5373.953,E2 -5373.953} C_VEL
LIN {X 0,Y 510.957,Z 662.089,A -85,B 0,C 180,E1 -5374.544,E2 -5374.544} C_VEL
LIN {X 0,Y 510.642,Z 673.107,A -85,B 0,C 180,E1 -5375.282,E2 -5375.282} C_VEL
LIN {X 0,Y 510.327,Z 683.26,A -85,B 0,C 180,E1 -5376.138,E2 -5376.138} C_VEL
LIN {X 0,Y 510.034,Z 692.51,A -85,B 0,C 180,E1 -5377.091,E2 -5377.091} C_VEL
LIN {X 0,Y 509.769,Z 700.893,A -85,B 0,C 180,E1 -5378.147,E2 -5378.147} C_VEL
LIN {X 0,Y 509.504,Z 709.121,A -85,B 0,C 180,E1 -5379.442,E2 -5379.442} C_VEL
LIN {X 0,Y 509.387,Z 715.301,A -85,B 0,C 180,E1 -5380.663,E2 -5380.663} C_VEL
LIN {X 0,Y 509.282,Z 720.394,A -85,B 0,C 180,E1 -5381.953,E2 -5381.953} C_VEL
LIN {X 0,Y 509.192,Z 723.944,A -85,B 0,C 180,E1 -5383.151,E2 -5383.151} C_VEL
LIN {X 0,Y 509.137,Z 725.818,A -85,B 0,C 180,E1 -5383.974,E2 -5383.974} C_VEL
LIN {X 0,Y 509.108,Z 727.613,A -85,B 0,C 180,E1 -5385.09,E2 -5385.09} C_VEL
LIN {X 0,Y 509.082,Z 728.677,A -85,B 0,C 180,E1 -5386.427,E2 -5386.427} C_VEL
LIN {X 0,Y 509.123,Z 728.807,A -85,B 0,C 180,E1 -5387.24,E2 -5387.24} C_VEL
LIN {X 0,Y 509.19,Z 728.118,A -85,B 0,C 180,E1 -5388.515,E2 -5388.515} C_VEL
LIN {X 0,Y 509.186,Z 726.638,A -85,B 0,C 180,E1 -5389.664,E2 -5389.664} C_VEL
LIN {X 0,Y 509.151,Z 725.117,A -85,B 0,C 180,E1 -5390.466,E2 -5390.466} C_VEL
LIN {X 0,Y 509.269,Z 721.941,A -85,B 0,C 180,E1 -5391.669,E2 -5391.669} C_VEL
LIN {X 0,Y 509.359,Z 717.731,A -85,B 0,C 180,E1 -5392.867,E2 -5392.867} C_VEL
LIN {X 0,Y 509.483,Z 711.353,A -85,B 0,C 180,E1 -5394.261,E2 -5394.261} C_VEL
LIN {X 0,Y 509.661,Z 704.324,A -85,B 0,C 180,E1 -5395.453,E2 -5395.453} C_VEL
LIN {X 0,Y 509.905,Z 695.669,A -85,B 0,C 180,E1 -5396.642,E2 -5396.642} C_VEL
LIN {X 0,Y 510.183,Z 686.725,A -85,B 0,C 180,E1 -5397.632,E2 -5397.632} C_VEL
LIN {X 0,Y 510.531,Z 676.835,A -85,B 0,C 180,E1 -5398.521,E2 -5398.521} C_VEL
LIN {X 0,Y 510.813,Z 666.006,A -85,B 0,C 180,E1 -5399.311,E2 -5399.311} C_VEL
LIN {X 0,Y 511.138,Z 653.805,A -85,B 0,C 180,E1 -5400,E2 -5400} C_VEL
LIN {X 0,Y 511.443,Z 640.829,A -85,B 0,C 180,E1 -5400.542,E2 -5400.542} C_VEL
LIN {X 0,Y 511.625,Z 627.882,A -85,B 0,C 180,E1 -5400.91,E2 -5400.91} C_VEL
LIN {X 0,Y 511.759,Z 601.096,A -85,B 0,C 180,E1 -5401.328,E2 -5401.328} C_VEL
LIN {X 0,Y 512.163,Z 527.079,A -85,B 0,C 180,E1 -5402.409,E2 -5402.409} C_VEL
LIN {X 0,Y 510.702,Z 517.919,A -85,B 0,C 180,E1 -5402.613,E2 -5402.613} C_VEL
LIN {X 0,Y 511.031,Z 496.302,A -85,B 0,C 180,E1 -5405.921,E2 -5405.921} C_VEL
LIN {X 0,Y 511.337,Z 479.559,A -85,B 0,C 180,E1 -5408.477,E2 -5408.477} C_VEL
LIN {X 0,Y 511.334,Z 468.83,A -85,B 0,C 180,E1 -5410.093,E2 -5410.093} C_VEL
LIN {X 0,Y 509.99,Z 461.076,A -85,B 0,C 180,E1 -5411.34,E2 -5411.34} C_VEL
LIN {X 0,Y 509.903,Z 460.973,A -85,B 0,C 180,E1 -5415.242,E2 -5415.242} C_VEL
LIN {X 0,Y 509.864,Z 460.974,A -85,B 0,C 180,E1 -5418.484,E2 -5418.484} C_VEL
LIN {X 0,Y 509.854,Z 460.979,A -85,B 0,C 180,E1 -5421.002,E2 -5421.002} C_VEL
LIN {X 0,Y 509.827,Z 460.977,A -85,B 0,C 180,E1 -5423.564,E2 -5423.564} C_VEL
LIN {X 0,Y 509.889,Z 460.97,A -85,B 0,C 180,E1 -5426.371,E2 -5426.371} C_VEL
LIN {X 0,Y 509.883,Z 460.975,A -85,B 0,C 180,E1 -5428.844,E2 -5428.844} C_VEL
LIN {X 0,Y 509.827,Z 460.975,A -85,B 0,C 180,E1 -5431.59,E2 -5431.59} C_VEL
LIN {X 0,Y 509.856,Z 460.975,A -85,B 0,C 180,E1 -5434.413,E2 -5434.413} C_VEL
LIN {X 0,Y 509.825,Z 460.976,A -85,B 0,C 180,E1 -5437.341,E2 -5437.341} C_VEL
LIN {X 0,Y 509.846,Z 460.978,A -85,B 0,C 180,E1 -5440.382,E2 -5440.382} C_VEL
LIN {X 0,Y 509.83,Z 460.977,A -85,B 0,C 180,E1 -5443.062,E2 -5443.062} C_VEL
LIN {X 0,Y 509.83,Z 460.976,A -85,B 0,C 180,E1 -5445.793,E2 -5445.793} C_VEL
LIN {X 0,Y 509.863,Z 460.977,A -85,B 0,C 180,E1 -5448.574,E2 -5448.574} C_VEL
LIN {X 0,Y 509.857,Z 460.965,A -85,B 0,C 180,E1 -5451.786,E2 -5451.786} C_VEL
LIN {X 0,Y 509.831,Z 460.975,A -85,B 0,C 180,E1 -5454.621,E2 -5454.621} C_VEL
LIN {X 0,Y 509.867,Z 460.974,A -85,B 0,C 180,E1 -5457.48,E2 -5457.48} C_VEL
LIN {X 0,Y 509.892,Z 461.001,A -85,B 0,C 180,E1 -5460.93,E2 -5460.93} C_VEL
LIN {X 0,Y 509.955,Z 461.429,A -85,B 0,C 180,E1 -5461.103,E2 -5461.103} C_VEL
LIN {X 0,Y 512.636,Z 473.801,A -85,B 0,C 180,E1 -5462.819,E2 -5462.819} C_VEL
LIN {X 0,Y 512.601,Z 483.051,A -85,B 0,C 180,E1 -5463.976,E2 -5463.976} C_VEL
LIN {X 0,Y 511.885,Z 508.978,A -85,B 0,C 180,E1 -5467.14,E2 -5467.14} C_VEL
LIN {X 0,Y 511.314,Z 532.043,A -85,B 0,C 180,E1 -5469.901,E2 -5469.901} C_VEL
LIN {X 0,Y 510.787,Z 556.504,A -85,B 0,C 180,E1 -5472.792,E2 -5472.792} C_VEL
LIN {X 0,Y 510.571,Z 570.314,A -85,B 0,C 180,E1 -5474.388,E2 -5474.388} C_VEL
LIN {X 0,Y 512.18,Z 585.057,A -85,B 0,C 180,E1 -5474.659,E2 -5474.659} C_VEL
LIN {X 0,Y 511.751,Z 680.578,A -85,B 0,C 180,E1 -5476.017,E2 -5476.017} C_VEL
LIN {X 0,Y 511.405,Z 693.997,A -85,B 0,C 180,E1 -5476.362,E2 -5476.362} C_VEL
LIN {X 0,Y 511.112,Z 707.446,A -85,B 0,C 180,E1 -5476.885,E2 -5476.885} C_VEL
LIN {X 0,Y 510.807,Z 719.131,A -85,B 0,C 180,E1 -5477.507,E2 -5477.507} C_VEL
LIN {X 0,Y 510.503,Z 730.539,A -85,B 0,C 180,E1 -5478.283,E2 -5478.283} C_VEL
LIN {X 0,Y 510.16,Z 741.158,A -85,B 0,C 180,E1 -5479.18,E2 -5479.18} C_VEL
LIN {X 0,Y 509.923,Z 749.866,A -85,B 0,C 180,E1 -5480.078,E2 -5480.078} C_VEL
LIN {X 0,Y 509.706,Z 757.916,A -85,B 0,C 180,E1 -5481.075,E2 -5481.075} C_VEL
LIN {X 0,Y 509.507,Z 765.794,A -85,B 0,C 180,E1 -5482.27,E2 -5482.27} C_VEL
LIN {X 0,Y 509.346,Z 773.07,A -85,B 0,C 180,E1 -5483.661,E2 -5483.661} C_VEL
LIN {X 0,Y 509.276,Z 777.919,A -85,B 0,C 180,E1 -5484.852,E2 -5484.852} C_VEL
LIN {X 0,Y 509.331,Z 781.643,A -85,B 0,C 180,E1 -5486.043,E2 -5486.043} C_VEL
LIN {X 0,Y 509.24,Z 783.531,A -85,B 0,C 180,E1 -5486.834,E2 -5486.834} C_VEL
LIN {X 0,Y 509.218,Z 784.983,A -85,B 0,C 180,E1 -5487.626,E2 -5487.626} C_VEL
LIN {X 0,Y 509.126,Z 786.619,A -85,B 0,C 180,E1 -5489.208,E2 -5489.208} C_VEL
LIN {X 0,Y 509.144,Z 786.843,A -85,B 0,C 180,E1 -5489.999,E2 -5489.999} C_VEL
LIN {X 0,Y 509.126,Z 786.627,A -85,B 0,C 180,E1 -5490.79,E2 -5490.79} C_VEL
LIN {X 0,Y 509.155,Z 786.011,A -85,B 0,C 180,E1 -5491.581,E2 -5491.581} C_VEL
LIN {X 0,Y 509.217,Z 784.996,A -85,B 0,C 180,E1 -5492.372,E2 -5492.372} C_VEL
LIN {X 0,Y 509.237,Z 783.559,A -85,B 0,C 180,E1 -5493.163,E2 -5493.163} C_VEL
LIN {X 0,Y 509.255,Z 780.537,A -85,B 0,C 180,E1 -5494.352,E2 -5494.352} C_VEL
LIN {X 0,Y 509.344,Z 776.486,A -85,B 0,C 180,E1 -5495.541,E2 -5495.541} C_VEL
LIN {X 0,Y 509.4,Z 770.694,A -85,B 0,C 180,E1 -5496.843,E2 -5496.843} C_VEL
LIN {X 0,Y 509.562,Z 763.411,A -85,B 0,C 180,E1 -5498.126,E2 -5498.126} C_VEL
LIN {X 0,Y 509.763,Z 754.951,A -85,B 0,C 180,E1 -5499.321,E2 -5499.321} C_VEL
LIN {X 0,Y 510.034,Z 746.309,A -85,B 0,C 180,E1 -5500.318,E2 -5500.318} C_VEL
LIN {X 0,Y 510.308,Z 735.646,A -85,B 0,C 180,E1 -5501.316,E2 -5501.316} C_VEL
LIN {X 0,Y 510.648,Z 723.859,A -85,B 0,C 180,E1 -5502.203,E2 -5502.203} C_VEL
LIN {X 0,Y 510.975,Z 711.668,A -85,B 0,C 180,E1 -5502.913,E2 -5502.913} C_VEL
LIN {X 0,Y 511.324,Z 699.215,A -85,B 0,C 180,E1 -5503.461,E2 -5503.461} C_VEL
LIN {X 0,Y 511.607,Z 686.458,A -85,B 0,C 180,E1 -5503.858,E2 -5503.858} C_VEL
LIN {X 0,Y 511.776,Z 671.353,A -85,B 0,C 180,E1 -5504.132,E2 -5504.132} C_VEL
LIN {X 0,Y 512.142,Z 584.017,A -85,B 0,C 180,E1 -5505.359,E2 -5505.359} C_VEL
LIN {X 0,Y 510.552,Z 570.331,A -85,B 0,C 180,E1 -5505.625,E2 -5505.625} C_VEL
LIN {X 0,Y 511.067,Z 544.683,A -85,B 0,C 180,E1 -5508.645,E2 -5508.645} C_VEL
LIN {X 0,Y 511.638,Z 518.594,A -85,B 0,C 180,E1 -5511.768,E2 -5511.768} C_VEL
LIN {X 0,Y 512.337,Z 495.992,A -85,B 0,C 180,E1 -5514.515,E2 -5514.515} C_VEL
LIN {X 0,Y 512.87,Z 474.821,A -85,B 0,C 180,E1 -5517.129,E2 -5517.129} C_VEL
LIN {X 0,Y 509.905,Z 461.097,A -85,B 0,C 180,E1 -5519.038,E2 -5519.038} C_VEL
LIN {X 0,Y 509.854,Z 460.977,A -85,B 0,C 180,E1 -5522.518,E2 -5522.518} C_VEL
LIN {X 0,Y 509.813,Z 460.979,A -85,B 0,C 180,E1 -5525.576,E2 -5525.576} C_VEL
LIN {X 0,Y 509.809,Z 460.982,A -85,B 0,C 180,E1 -5528.34,E2 -5528.34} C_VEL
LIN {X 0,Y 509.823,Z 460.974,A -85,B 0,C 180,E1 -5531.427,E2 -5531.427} C_VEL
LIN {X 0,Y 509.83,Z 460.976,A -85,B 0,C 180,E1 -5534.669,E2 -5534.669} C_VEL
LIN {X 0,Y 509.836,Z 460.979,A -85,B 0,C 180,E1 -5538.103,E2 -5538.103} C_VEL
LIN {X 0,Y 509.822,Z 460.977,A -85,B 0,C 180,E1 -5540.645,E2 -5540.645} C_VEL
LIN {X 0,Y 509.798,Z 460.978,A -85,B 0,C 180,E1 -5543.644,E2 -5543.644} C_VEL
LIN {X 0,Y 509.847,Z 460.976,A -85,B 0,C 180,E1 -5546.538,E2 -5546.538} C_VEL
LIN {X 0,Y 509.831,Z 460.973,A -85,B 0,C 180,E1 -5549.333,E2 -5549.333} C_VEL
LIN {X 0,Y 509.871,Z 460.973,A -85,B 0,C 180,E1 -5552.053,E2 -5552.053} C_VEL
LIN {X 0,Y 509.805,Z 460.98,A -85,B 0,C 180,E1 -5554.7,E2 -5554.7} C_VEL
LIN {X 0,Y 509.812,Z 460.975,A -85,B 0,C 180,E1 -5557.457,E2 -5557.457} C_VEL
LIN {X 0,Y 509.903,Z 460.966,A -85,B 0,C 180,E1 -5559.844,E2 -5559.844} C_VEL
LIN {X 0,Y 509.864,Z 460.969,A -85,B 0,C 180,E1 -5563.174,E2 -5563.174} C_VEL
LIN {X 0,Y 509.844,Z 460.971,A -85,B 0,C 180,E1 -5565.633,E2 -5565.633} C_VEL
LIN {X 0,Y 509.905,Z 460.967,A -85,B 0,C 180,E1 -5568.874,E2 -5568.874} C_VEL
LIN {X 0,Y 509.936,Z 460.963,A -85,B 0,C 180,E1 -5572.078,E2 -5572.078} C_VEL
LIN {X 0,Y 509.961,Z 460.965,A -85,B 0,C 180,E1 -5574.464,E2 -5574.464} C_VEL
LIN {X 0,Y 510.037,Z 460.947,A -85,B 0,C 180,E1 -5577.631,E2 -5577.631} C_VEL
LIN {X 0,Y 510.052,Z 460.951,A -85,B 0,C 180,E1 -5580.789,E2 -5580.789} C_VEL
LIN {X 0,Y 509.942,Z 460.96,A -85,B 0,C 180,E1 -5583.16,E2 -5583.16} C_VEL
LIN {X 0,Y 509.938,Z 460.965,A -85,B 0,C 180,E1 -5586.33,E2 -5586.33} C_VEL
LIN {X 0,Y 509.905,Z 460.971,A -85,B 0,C 180,E1 -5588.72,E2 -5588.72} C_VEL
LIN {X 0,Y 509.891,Z 460.966,A -85,B 0,C 180,E1 -5591.932,E2 -5591.932} C_VEL
LIN {X 0,Y 509.879,Z 460.968,A -85,B 0,C 180,E1 -5595.242,E2 -5595.242} C_VEL
LIN {X 0,Y 509.874,Z 460.968,A -85,B 0,C 180,E1 -5598.001,E2 -5598.001} C_VEL
LIN {X 0,Y 509.837,Z 460.977,A -85,B 0,C 180,E1 -5601.002,E2 -5601.002} C_VEL
LIN {X 0,Y 509.823,Z 460.974,A -85,B 0,C 180,E1 -5603.563,E2 -5603.563} C_VEL
LIN {X 0,Y 509.898,Z 460.968,A -85,B 0,C 180,E1 -5606.379,E2 -5606.379} C_VEL
LIN {X 0,Y 509.864,Z 460.977,A -85,B 0,C 180,E1 -5608.845,E2 -5608.845} C_VEL
LIN {X 0,Y 509.812,Z 460.975,A -85,B 0,C 180,E1 -5611.59,E2 -5611.59} C_VEL
LIN {X 0,Y 509.842,Z 460.975,A -85,B 0,C 180,E1 -5614.414,E2 -5614.414} C_VEL
LIN {X 0,Y 509.806,Z 460.978,A -85,B 0,C 180,E1 -5617.341,E2 -5617.341} C_VEL
LIN {X 0,Y 509.826,Z 460.976,A -85,B 0,C 180,E1 -5620.383,E2 -5620.383} C_VEL
LIN {X 0,Y 509.828,Z 460.979,A -85,B 0,C 180,E1 -5623.065,E2 -5623.065} C_VEL
LIN {X 0,Y 509.82,Z 460.974,A -85,B 0,C 180,E1 -5625.793,E2 -5625.793} C_VEL
LIN {X 0,Y 509.861,Z 460.973,A -85,B 0,C 180,E1 -5628.577,E2 -5628.577} C_VEL
LIN {X 0,Y 509.846,Z 460.971,A -85,B 0,C 180,E1 -5631.787,E2 -5631.787} C_VEL
LIN {X 0,Y 509.82,Z 460.974,A -85,B 0,C 180,E1 -5633.754,E2 -5633.754} C_VEL
LIN {X 0,Y 509.154,Z 461.06,A -85,B 0,C 180,E1 -5634.414,E2 -5634.414} C_VEL
LIN {X 0,Y 506.336,Z 461.416,A -85,B 0,C 180,E1 -5635.485,E2 -5635.485} C_VEL
LIN {X 0,Y 503.944,Z 461.717,A -85,B 0,C 180,E1 -5636.349,E2 -5636.349} C_VEL
LIN {X 0,Y 502.896,Z 461.845,A -85,B 0,C 180,E1 -5637.015,E2 -5637.015} C_VEL
LIN {X 0,Y 502.799,Z 461.854,A -85,B 0,C 180,E1 -5637.241,E2 -5637.241} C_VEL
LIN {X 0,Y 502.807,Z 461.848,A -85,B 0,C 180,E1 -5640.066,E2 -5640.066} C_VEL
LIN {X 0,Y 502.827,Z 461.848,A -85,B 0,C 180,E1 -5642.535,E2 -5642.535} C_VEL
LIN {X 0,Y 502.822,Z 461.851,A -85,B 0,C 180,E1 -5645.3,E2 -5645.3} C_VEL
LIN {X 0,Y 502.787,Z 461.851,A -85,B 0,C 180,E1 -5647.828,E2 -5647.828} C_VEL
LIN {X 0,Y 502.82,Z 461.847,A -85,B 0,C 180,E1 -5650.402,E2 -5650.402} C_VEL
LIN {X 0,Y 502.83,Z 461.852,A -85,B 0,C 180,E1 -5652.933,E2 -5652.933} C_VEL
LIN {X 0,Y 502.841,Z 461.848,A -85,B 0,C 180,E1 -5655.431,E2 -5655.431} C_VEL
LIN {X 0,Y 502.874,Z 461.843,A -85,B 0,C 180,E1 -5658.718,E2 -5658.718} C_VEL
LIN {X 0,Y 502.899,Z 461.839,A -85,B 0,C 180,E1 -5661.968,E2 -5661.968} C_VEL
LIN {X 0,Y 502.939,Z 461.835,A -85,B 0,C 180,E1 -5664.388,E2 -5664.388} C_VEL
LIN {X 0,Y 503.025,Z 461.828,A -85,B 0,C 180,E1 -5667.599,E2 -5667.599} C_VEL
LIN {X 0,Y 502.933,Z 462.04,A -85,B 0,C 180,E1 -5668.52,E2 -5668.52} C_VEL
LIN {X 0,Y 503.191,Z 463.173,A -85,B 0,C 180,E1 -5668.652,E2 -5668.652} C_VEL
LIN {X 0,Y 505.427,Z 469.365,A -85,B 0,C 180,E1 -5668.821,E2 -5668.821} C_VEL
LIN {X 0,Y 505.152,Z 543.059,A -85,B 0,C 180,E1 -5669.902,E2 -5669.902} C_VEL
LIN {X 0,Y 505.048,Z 555.901,A -85,B 0,C 180,E1 -5670.25,E2 -5670.25} C_VEL
LIN {X 0,Y 504.903,Z 568.301,A -85,B 0,C 180,E1 -5670.749,E2 -5670.749} C_VEL
LIN {X 0,Y 504.665,Z 580.198,A -85,B 0,C 180,E1 -5671.398,E2 -5671.398} C_VEL
LIN {X 0,Y 504.37,Z 591.496,A -85,B 0,C 180,E1 -5672.197,E2 -5672.197} C_VEL
LIN {X 0,Y 504.002,Z 601.713,A -85,B 0,C 180,E1 -5673.099,E2 -5673.099} C_VEL
LIN {X 0,Y 503.76,Z 610.048,A -85,B 0,C 180,E1 -5674.001,E2 -5674.001} C_VEL
LIN {X 0,Y 503.473,Z 617.768,A -85,B 0,C 180,E1 -5675.006,E2 -5675.006} C_VEL
LIN {X 0,Y 503.265,Z 625.301,A -85,B 0,C 180,E1 -5676.214,E2 -5676.214} C_VEL
LIN {X 0,Y 503.004,Z 632.086,A -85,B 0,C 180,E1 -5677.589,E2 -5677.589} C_VEL
LIN {X 0,Y 502.824,Z 636.908,A -85,B 0,C 180,E1 -5678.845,E2 -5678.845} C_VEL
LIN {X 0,Y 502.692,Z 640.46,A -85,B 0,C 180,E1 -5680.066,E2 -5680.066} C_VEL
LIN {X 0,Y 502.615,Z 643.006,A -85,B 0,C 180,E1 -5681.29,E2 -5681.29} C_VEL
LIN {X 0,Y 502.581,Z 644.201,A -85,B 0,C 180,E1 -5682.109,E2 -5682.109} C_VEL
LIN {X 0,Y 502.519,Z 644.953,A -85,B 0,C 180,E1 -5682.932,E2 -5682.932} C_VEL
LIN {X 0,Y 502.514,Z 645.272,A -85,B 0,C 180,E1 -5684.582,E2 -5684.582} C_VEL
LIN {X 0,Y 502.552,Z 644.813,A -85,B 0,C 180,E1 -5685.41,E2 -5685.41} C_VEL
LIN {X 0,Y 502.58,Z 643.916,A -85,B 0,C 180,E1 -5686.242,E2 -5686.242} C_VEL
LIN {X 0,Y 502.605,Z 642.612,A -85,B 0,C 180,E1 -5687.078,E2 -5687.078} C_VEL
LIN {X 0,Y 502.729,Z 640.433,A -85,B 0,C 180,E1 -5688.082,E2 -5688.082} C_VEL
LIN {X 0,Y 502.888,Z 635.861,A -85,B 0,C 180,E1 -5689.599,E2 -5689.599} C_VEL
LIN {X 0,Y 503.129,Z 629.715,A -85,B 0,C 180,E1 -5691.07,E2 -5691.07} C_VEL
LIN {X 0,Y 503.377,Z 622.876,A -85,B 0,C 180,E1 -5692.338,E2 -5692.338} C_VEL
LIN {X 0,Y 503.646,Z 615.545,A -85,B 0,C 180,E1 -5693.435,E2 -5693.435} C_VEL
LIN {X 0,Y 503.967,Z 606.714,A -85,B 0,C 180,E1 -5694.513,E2 -5694.513} C_VEL
LIN {X 0,Y 504.267,Z 596.569,A -85,B 0,C 180,E1 -5695.509,E2 -5695.509} C_VEL
LIN {X 0,Y 504.599,Z 585.795,A -85,B 0,C 180,E1 -5696.358,E2 -5696.358} C_VEL
LIN {X 0,Y 504.895,Z 573.885,A -85,B 0,C 180,E1 -5697.092,E2 -5697.092} C_VEL
LIN {X 0,Y 505.062,Z 561.311,A -85,B 0,C 180,E1 -5697.674,E2 -5697.674} C_VEL
LIN {X 0,Y 505.191,Z 548.535,A -85,B 0,C 180,E1 -5698.089,E2 -5698.089} C_VEL
LIN {X 0,Y 505.205,Z 535.046,A -85,B 0,C 180,E1 -5698.349,E2 -5698.349} C_VEL
LIN {X 0,Y 505.43,Z 469.491,A -85,B 0,C 180,E1 -5699.303,E2 -5699.303} C_VEL
LIN {X 0,Y 502.994,Z 462.676,A -85,B 0,C 180,E1 -5699.516,E2 -5699.516} C_VEL
LIN {X 0,Y 502.835,Z 461.905,A -85,B 0,C 180,E1 -5699.691,E2 -5699.691} C_VEL
LIN {X 0,Y 502.832,Z 461.851,A -85,B 0,C 180,E1 -5703.032,E2 -5703.032} C_VEL
LIN {X 0,Y 502.777,Z 461.855,A -85,B 0,C 180,E1 -5705.952,E2 -5705.952} C_VEL
LIN {X 0,Y 502.804,Z 461.853,A -85,B 0,C 180,E1 -5708.977,E2 -5708.977} C_VEL
LIN {X 0,Y 502.799,Z 461.85,A -85,B 0,C 180,E1 -5712.14,E2 -5712.14} C_VEL
LIN {X 0,Y 502.79,Z 461.853,A -85,B 0,C 180,E1 -5715.471,E2 -5715.471} C_VEL
LIN {X 0,Y 502.824,Z 461.855,A -85,B 0,C 180,E1 -5718.935,E2 -5718.935} C_VEL
LIN {X 0,Y 502.806,Z 461.853,A -85,B 0,C 180,E1 -5722.048,E2 -5722.048} C_VEL
LIN {X 0,Y 502.833,Z 462.086,A -85,B 0,C 180,E1 -5722.448,E2 -5722.448} C_VEL
LIN {X 0,Y 504.545,Z 470.632,A -85,B 0,C 180,E1 -5723.893,E2 -5723.893} C_VEL
LIN {X 0,Y 504.447,Z 481.796,A -85,B 0,C 180,E1 -5725.65,E2 -5725.65} C_VEL
LIN {X 0,Y 504.047,Z 498.443,A -85,B 0,C 180,E1 -5728.271,E2 -5728.271} C_VEL
LIN {X 0,Y 503.636,Z 517.598,A -85,B 0,C 180,E1 -5731.248,E2 -5731.248} C_VEL
LIN {X 0,Y 505.449,Z 529.099,A -85,B 0,C 180,E1 -5731.503,E2 -5731.503} C_VEL
LIN {X 0,Y 504.789,Z 626.396,A -85,B 0,C 180,E1 -5732.957,E2 -5732.957} C_VEL
LIN {X 0,Y 504.541,Z 639.457,A -85,B 0,C 180,E1 -5733.31,E2 -5733.31} C_VEL
LIN {X 0,Y 504.247,Z 651.381,A -85,B 0,C 180,E1 -5733.791,E2 -5733.791} C_VEL
LIN {X 0,Y 503.943,Z 664.175,A -85,B 0,C 180,E1 -5734.488,E2 -5734.488} C_VEL
LIN {X 0,Y 503.634,Z 674.984,A -85,B 0,C 180,E1 -5735.252,E2 -5735.252} C_VEL
LIN {X 0,Y 503.279,Z 684.789,A -85,B 0,C 180,E1 -5736.111,E2 -5736.111} C_VEL
LIN {X 0,Y 502.968,Z 694.746,A -85,B 0,C 180,E1 -5737.185,E2 -5737.185} C_VEL
LIN {X 0,Y 502.697,Z 702.785,A -85,B 0,C 180,E1 -5738.255,E2 -5738.255} C_VEL
LIN {X 0,Y 502.435,Z 710.517,A -85,B 0,C 180,E1 -5739.532,E2 -5739.532} C_VEL
LIN {X 0,Y 502.322,Z 716.645,A -85,B 0,C 180,E1 -5740.805,E2 -5740.805} C_VEL
LIN {X 0,Y 502.173,Z 721.509,A -85,B 0,C 180,E1 -5742.117,E2 -5742.117} C_VEL
LIN {X 0,Y 502.129,Z 723.825,A -85,B 0,C 180,E1 -5742.907,E2 -5742.907} C_VEL
LIN {X 0,Y 502.067,Z 725.804,A -85,B 0,C 180,E1 -5743.742,E2 -5743.742} C_VEL
LIN {X 0,Y 502.049,Z 727.915,A -85,B 0,C 180,E1 -5744.999,E2 -5744.999} C_VEL
LIN {X 0,Y 502.004,Z 729.013,A -85,B 0,C 180,E1 -5746.232,E2 -5746.232} C_VEL
LIN {X 0,Y 502.02,Z 729.233,A -85,B 0,C 180,E1 -5747.057,E2 -5747.057} C_VEL
LIN {X 0,Y 502.114,Z 728.594,A -85,B 0,C 180,E1 -5748.462,E2 -5748.462} C_VEL
LIN {X 0,Y 502.13,Z 727.35,A -85,B 0,C 180,E1 -5749.517,E2 -5749.517} C_VEL
LIN {X 0,Y 502.07,Z 725.901,A -85,B 0,C 180,E1 -5750.33,E2 -5750.33} C_VEL
LIN {X 0,Y 502.212,Z 722.878,A -85,B 0,C 180,E1 -5751.551,E2 -5751.551} C_VEL
LIN {X 0,Y 502.293,Z 718.818,A -85,B 0,C 180,E1 -5752.766,E2 -5752.766} C_VEL
LIN {X 0,Y 502.408,Z 712.628,A -85,B 0,C 180,E1 -5754.179,E2 -5754.179} C_VEL
LIN {X 0,Y 502.596,Z 705.846,A -85,B 0,C 180,E1 -5755.388,E2 -5755.388} C_VEL
LIN {X 0,Y 502.822,Z 697.394,A -85,B 0,C 180,E1 -5756.595,E2 -5756.595} C_VEL
LIN {X 0,Y 503.148,Z 688.738,A -85,B 0,C 180,E1 -5757.599,E2 -5757.599} C_VEL
LIN {X 0,Y 503.467,Z 679.264,A -85,B 0,C 180,E1 -5758.5,E2 -5758.5} C_VEL
LIN {X 0,Y 503.801,Z 668.844,A -85,B 0,C 180,E1 -5759.301,E2 -5759.301} C_VEL
LIN {X 0,Y 504.087,Z 657.378,A -85,B 0,C 180,E1 -5760,E2 -5760} C_VEL
LIN {X 0,Y 504.445,Z 645.591,A -85,B 0,C 180,E1 -5760.549,E2 -5760.549} C_VEL
LIN {X 0,Y 504.652,Z 632.809,A -85,B 0,C 180,E1 -5760.973,E2 -5760.973} C_VEL
LIN {X 0,Y 504.793,Z 619.412,A -85,B 0,C 180,E1 -5761.247,E2 -5761.247} C_VEL
LIN {X 0,Y 505.366,Z 528.238,A -85,B 0,C 180,E1 -5762.603,E2 -5762.603} C_VEL
LIN {X 0,Y 503.795,Z 518.374,A -85,B 0,C 180,E1 -5762.824,E2 -5762.824} C_VEL
LIN {X 0,Y 503.884,Z 508.005,A -85,B 0,C 180,E1 -5764.4,E2 -5764.4} C_VEL
LIN {X 0,Y 504.299,Z 491.25,A -85,B 0,C 180,E1 -5767.004,E2 -5767.004} C_VEL
LIN {X 0,Y 504.511,Z 471.237,A -85,B 0,C 180,E1 -5770.028,E2 -5770.028} C_VEL
LIN {X 0,Y 502.925,Z 461.936,A -85,B 0,C 180,E1 -5771.537,E2 -5771.537} C_VEL
LIN {X 0,Y 502.846,Z 461.852,A -85,B 0,C 180,E1 -5775.336,E2 -5775.336} C_VEL
LIN {X 0,Y 502.829,Z 461.853,A -85,B 0,C 180,E1 -5778.752,E2 -5778.752} C_VEL
LIN {X 0,Y 502.789,Z 461.857,A -85,B 0,C 180,E1 -5781.311,E2 -5781.311} C_VEL
LIN {X 0,Y 502.777,Z 461.854,A -85,B 0,C 180,E1 -5783.915,E2 -5783.915} C_VEL
LIN {X 0,Y 502.844,Z 461.85,A -85,B 0,C 180,E1 -5786.568,E2 -5786.568} C_VEL
LIN {X 0,Y 502.831,Z 461.849,A -85,B 0,C 180,E1 -5789.288,E2 -5789.288} C_VEL
LIN {X 0,Y 502.791,Z 461.852,A -85,B 0,C 180,E1 -5792.084,E2 -5792.084} C_VEL
LIN {X 0,Y 502.807,Z 461.854,A -85,B 0,C 180,E1 -5794.965,E2 -5794.965} C_VEL
LIN {X 0,Y 502.801,Z 461.851,A -85,B 0,C 180,E1 -5797.954,E2 -5797.954} C_VEL
LIN {X 0,Y 502.828,Z 461.85,A -85,B 0,C 180,E1 -5801.066,E2 -5801.066} C_VEL
LIN {X 0,Y 502.794,Z 461.857,A -85,B 0,C 180,E1 -5804.529,E2 -5804.529} C_VEL
LIN {X 0,Y 502.803,Z 461.853,A -85,B 0,C 180,E1 -5807.86,E2 -5807.86} C_VEL
LIN {X 0,Y 502.79,Z 461.854,A -85,B 0,C 180,E1 -5810.246,E2 -5810.246} C_VEL
LIN {X 0,Y 502.761,Z 461.856,A -85,B 0,C 180,E1 -5813.051,E2 -5813.051} C_VEL
LIN {X 0,Y 502.793,Z 461.848,A -85,B 0,C 180,E1 -5816.004,E2 -5816.004} C_VEL
LIN {X 0,Y 502.801,Z 461.854,A -85,B 0,C 180,E1 -5818.856,E2 -5818.856} C_VEL
LIN {X 0,Y 502.903,Z 462.086,A -85,B 0,C 180,E1 -5820.838,E2 -5820.838} C_VEL
LIN {X 0,Y 505.818,Z 475.807,A -85,B 0,C 180,E1 -5822.778,E2 -5822.778} C_VEL
LIN {X 0,Y 505.501,Z 490.626,A -85,B 0,C 180,E1 -5824.649,E2 -5824.649} C_VEL
LIN {X 0,Y 504.801,Z 515.37,A -85,B 0,C 180,E1 -5827.703,E2 -5827.703} C_VEL
LIN {X 0,Y 504.091,Z 541.526,A -85,B 0,C 180,E1 -5830.873,E2 -5830.873} C_VEL
LIN {X 0,Y 503.552,Z 565.916,A -85,B 0,C 180,E1 -5833.79,E2 -5833.79} C_VEL
LIN {X 0,Y 503.509,Z 569.155,A -85,B 0,C 180,E1 -5834.157,E2 -5834.157} C_VEL
LIN {X 0,Y 505.311,Z 586.045,A -85,B 0,C 180,E1 -5834.474,E2 -5834.474} C_VEL
LIN {X 0,Y 504.823,Z 679.514,A -85,B 0,C 180,E1 -5835.821,E2 -5835.821} C_VEL
LIN {X 0,Y 504.493,Z 692.182,A -85,B 0,C 180,E1 -5836.146,E2 -5836.146} C_VEL
LIN {X 0,Y 504.166,Z 705.264,A -85,B 0,C 180,E1 -5836.65,E2 -5836.65} C_VEL
LIN {X 0,Y 503.859,Z 717.271,A -85,B 0,C 180,E1 -5837.28,E2 -5837.28} C_VEL
LIN {X 0,Y 503.558,Z 728.197,A -85,B 0,C 180,E1 -5838.017,E2 -5838.017} C_VEL
LIN {X 0,Y 503.114,Z 739.032,A -85,B 0,C 180,E1 -5838.925,E2 -5838.925} C_VEL
LIN {X 0,Y 502.872,Z 748.841,A -85,B 0,C 180,E1 -5839.938,E2 -5839.938} C_VEL
LIN {X 0,Y 502.654,Z 756.897,A -85,B 0,C 180,E1 -5840.949,E2 -5840.949} C_VEL
LIN {X 0,Y 502.422,Z 764.777,A -85,B 0,C 180,E1 -5842.16,E2 -5842.16} C_VEL
LIN {X 0,Y 502.288,Z 771.418,A -85,B 0,C 180,E1 -5843.431,E2 -5843.431} C_VEL
LIN {X 0,Y 502.237,Z 776.914,A -85,B 0,C 180,E1 -5844.78,E2 -5844.78} C_VEL
LIN {X 0,Y 502.268,Z 780.65,A -85,B 0,C 180,E1 -5845.987,E2 -5845.987} C_VEL
LIN {X 0,Y 502.198,Z 782.531,A -85,B 0,C 180,E1 -5846.79,E2 -5846.79} C_VEL
LIN {X 0,Y 502.177,Z 783.988,A -85,B 0,C 180,E1 -5847.592,E2 -5847.592} C_VEL
LIN {X 0,Y 502.121,Z 785.018,A -85,B 0,C 180,E1 -5848.395,E2 -5848.395} C_VEL
LIN {X 0,Y 502.133,Z 785.863,A -85,B 0,C 180,E1 -5849.999,E2 -5849.999} C_VEL
LIN {X 0,Y 502.092,Z 785.651,A -85,B 0,C 180,E1 -5850.801,E2 -5850.801} C_VEL
LIN {X 0,Y 502.119,Z 785.038,A -85,B 0,C 180,E1 -5851.603,E2 -5851.603} C_VEL
LIN {X 0,Y 502.173,Z 784.02,A -85,B 0,C 180,E1 -5852.405,E2 -5852.405} C_VEL
LIN {X 0,Y 502.193,Z 782.578,A -85,B 0,C 180,E1 -5853.208,E2 -5853.208} C_VEL
LIN {X 0,Y 502.195,Z 779.542,A -85,B 0,C 180,E1 -5854.413,E2 -5854.413} C_VEL
LIN {X 0,Y 502.284,Z 775.502,A -85,B 0,C 180,E1 -5855.619,E2 -5855.619} C_VEL
LIN {X 0,Y 502.331,Z 769.352,A -85,B 0,C 180,E1 -5857.01,E2 -5857.01} C_VEL
LIN {X 0,Y 502.493,Z 762.428,A -85,B 0,C 180,E1 -5858.241,E2 -5858.241} C_VEL
LIN {X 0,Y 502.713,Z 753.962,A -85,B 0,C 180,E1 -5859.453,E2 -5859.453} C_VEL
LIN {X 0,Y 502.997,Z 745.318,A -85,B 0,C 180,E1 -5860.464,E2 -5860.464} C_VEL
LIN {X 0,Y 503.269,Z 734.65,A -85,B 0,C 180,E1 -5861.477,E2 -5861.477} C_VEL
LIN {X 0,Y 503.597,Z 724.117,A -85,B 0,C 180,E1 -5862.287,E2 -5862.287} C_VEL
LIN {X 0,Y 503.934,Z 712.621,A -85,B 0,C 180,E1 -5862.995,E2 -5862.995} C_VEL
LIN {X 0,Y 504.312,Z 700.834,A -85,B 0,C 180,E1 -5863.549,E2 -5863.549} C_VEL
LIN {X 0,Y 504.652,Z 687.291,A -85,B 0,C 180,E1 -5864.001,E2 -5864.001} C_VEL
LIN {X 0,Y 504.854,Z 673.901,A -85,B 0,C 180,E1 -5864.278,E2 -5864.278} C_VEL
LIN {X 0,Y 505.191,Z 584.112,A -85,B 0,C 180,E1 -5865.56,E2 -5865.56} C_VEL
LIN {X 0,Y 503.505,Z 569.435,A -85,B 0,C 180,E1 -5865.842,E2 -5865.842} C_VEL
LIN {X 0,Y 504.028,Z 545.455,A -85,B 0,C 180,E1 -5868.704,E2 -5868.704} C_VEL
LIN {X 0,Y 504.636,Z 521.181,A -85,B 0,C 180,E1 -5871.656,E2 -5871.656} C_VEL
LIN {X 0,Y 505.397,Z 496.833,A -85,B 0,C 180,E1 -5874.655,E2 -5874.655} C_VEL
LIN {X 0,Y 505.938,Z 476.169,A -85,B 0,C 180,E1 -5877.248,E2 -5877.248} C_VEL
LIN {X 0,Y 502.868,Z 462.004,A -85,B 0,C 180,E1 -5879.23,E2 -5879.23} C_VEL
LIN {X 0,Y 502.777,Z 461.861,A -85,B 0,C 180,E1 -5882.083,E2 -5882.083} C_VEL
LIN {X 0,Y 502.786,Z 461.853,A -85,B 0,C 180,E1 -5884.965,E2 -5884.965} C_VEL
LIN {X 0,Y 502.757,Z 461.859,A -85,B 0,C 180,E1 -5888.48,E2 -5888.48} C_VEL
LIN {X 0,Y 502.763,Z 461.853,A -85,B 0,C 180,E1 -5891.069,E2 -5891.069} C_VEL
LIN {X 0,Y 502.744,Z 461.856,A -85,B 0,C 180,E1 -5893.371,E2 -5893.371} C_VEL
LIN {X 0,Y 502.769,Z 461.854,A -85,B 0,C 180,E1 -5895.659,E2 -5895.659} C_VEL
LIN {X 0,Y 502.785,Z 461.854,A -85,B 0,C 180,E1 -5897.859,E2 -5897.859} C_VEL
LIN {X 0,Y 502.783,Z 461.851,A -85,B 0,C 180,E1 -5901.022,E2 -5901.022} C_VEL
LIN {X 0,Y 502.76,Z 461.861,A -85,B 0,C 180,E1 -5904.168,E2 -5904.168} C_VEL
LIN {X 0,Y 502.821,Z 461.847,A -85,B 0,C 180,E1 -5906.992,E2 -5906.992} C_VEL
LIN {X 0,Y 502.802,Z 461.853,A -85,B 0,C 180,E1 -5910.064,E2 -5910.064} C_VEL
LIN {X 0,Y 502.811,Z 461.854,A -85,B 0,C 180,E1 -5912.532,E2 -5912.532} C_VEL
LIN {X 0,Y 502.765,Z 461.853,A -85,B 0,C 180,E1 -5915.31,E2 -5915.31} C_VEL
LIN {X 0,Y 502.766,Z 461.855,A -85,B 0,C 180,E1 -5917.825,E2 -5917.825} C_VEL
LIN {X 0,Y 502.808,Z 461.857,A -85,B 0,C 180,E1 -5920.399,E2 -5920.399} C_VEL
LIN {X 0,Y 502.813,Z 461.849,A -85,B 0,C 180,E1 -5922.931,E2 -5922.931} C_VEL
LIN {X 0,Y 502.827,Z 461.845,A -85,B 0,C 180,E1 -5925.428,E2 -5925.428} C_VEL
LIN {X 0,Y 502.868,Z 461.845,A -85,B 0,C 180,E1 -5928.716,E2 -5928.716} C_VEL
LIN {X 0,Y 502.886,Z 461.84,A -85,B 0,C 180,E1 -5931.966,E2 -5931.966} C_VEL
LIN {X 0,Y 502.915,Z 461.842,A -85,B 0,C 180,E1 -5934.386,E2 -5934.386} C_VEL
LIN {X 0,Y 503.007,Z 461.823,A -85,B 0,C 180,E1 -5937.597,E2 -5937.597} C_VEL
LIN {X 0,Y 503.009,Z 461.824,A -85,B 0,C 180,E1 -5940,E2 -5940} C_VEL
LIN {X 0,Y 503.009,Z 461.829,A -85,B 0,C 180,E1 -5942.402,E2 -5942.402} C_VEL
LIN {X 0,Y 502.92,Z 461.834,A -85,B 0,C 180,E1 -5945.613,E2 -5945.613} C_VEL
LIN {X 0,Y 502.888,Z 461.839,A -85,B 0,C 180,E1 -5948.033,E2 -5948.033} C_VEL
LIN {X 0,Y 502.867,Z 461.841,A -85,B 0,C 180,E1 -5951.283,E2 -5951.283} C_VEL
LIN {X 0,Y 502.837,Z 461.852,A -85,B 0,C 180,E1 -5954.571,E2 -5954.571} C_VEL
LIN {X 0,Y 502.847,Z 461.843,A -85,B 0,C 180,E1 -5957.907,E2 -5957.907} C_VEL
LIN {X 0,Y 502.815,Z 461.853,A -85,B 0,C 180,E1 -5960.537,E2 -5960.537} C_VEL
LIN {X 0,Y 502.783,Z 461.855,A -85,B 0,C 180,E1 -5963.041,E2 -5963.041} C_VEL
LIN {X 0,Y 502.826,Z 461.845,A -85,B 0,C 180,E1 -5965.676,E2 -5965.676} C_VEL
LIN {X 0,Y 502.827,Z 461.849,A -85,B 0,C 180,E1 -5968.373,E2 -5968.373} C_VEL
LIN {X 0,Y 502.783,Z 461.851,A -85,B 0,C 180,E1 -5971.5,E2 -5971.5} C_VEL
LIN {X 0,Y 502.794,Z 461.853,A -85,B 0,C 180,E1 -5974.446,E2 -5974.446} C_VEL
LIN {X 0,Y 502.768,Z 461.856,A -85,B 0,C 180,E1 -5977.179,E2 -5977.179} C_VEL
LIN {X 0,Y 502.776,Z 461.852,A -85,B 0,C 180,E1 -5980.016,E2 -5980.016} C_VEL
LIN {X 0,Y 502.791,Z 461.851,A -85,B 0,C 180,E1 -5982.2,E2 -5982.2} C_VEL
LIN {X 0,Y 502.789,Z 461.852,A -85,B 0,C 180,E1 -5985.469,E2 -5985.469} C_VEL
LIN {X 0,Y 502.828,Z 461.845,A -85,B 0,C 180,E1 -5987.866,E2 -5987.866} C_VEL
LIN {X 0,Y 502.812,Z 461.855,A -85,B 0,C 180,E1 -5991.027,E2 -5991.027} C_VEL
LIN {X 0,Y 502.773,Z 461.852,A -85,B 0,C 180,E1 -5994.169,E2 -5994.169} C_VEL
LIN {X 0,Y 502.799,Z 461.854,A -85,B 0,C 180,E1 -5997.241,E2 -5997.241} C_VEL
LIN {X 0,Y 502.1,Z 461.938,A -85,B 0,C 180,E1 -5997.91,E2 -5997.91} C_VEL
LIN {X 0,Y 499.235,Z 462.302,A -85,B 0,C 180,E1 -5998.995,E2 -5998.995} C_VEL
LIN {X 0,Y 496.839,Z 462.595,A -85,B 0,C 180,E1 -5999.87,E2 -5999.87} C_VEL
LIN {X 0,Y 495.823,Z 462.721,A -85,B 0,C 180,E1 -6000.546,E2 -6000.546} C_VEL
LIN {X 0,Y 495.746,Z 462.729,A -85,B 0,C 180,E1 -6000.775,E2 -6000.775} C_VEL
LIN {X 0,Y 495.784,Z 462.723,A -85,B 0,C 180,E1 -6003.934,E2 -6003.934} C_VEL
LIN {X 0,Y 495.752,Z 462.734,A -85,B 0,C 180,E1 -6007.141,E2 -6007.141} C_VEL
LIN {X 0,Y 495.772,Z 462.724,A -85,B 0,C 180,E1 -6010.111,E2 -6010.111} C_VEL
LIN {X 0,Y 495.782,Z 462.726,A -85,B 0,C 180,E1 -6012.683,E2 -6012.683} C_VEL
LIN {X 0,Y 495.786,Z 462.73,A -85,B 0,C 180,E1 -6015.219,E2 -6015.219} C_VEL
LIN {X 0,Y 495.848,Z 462.716,A -85,B 0,C 180,E1 -6018.556,E2 -6018.556} C_VEL
LIN {X 0,Y 495.871,Z 462.715,A -85,B 0,C 180,E1 -6021.853,E2 -6021.853} C_VEL
LIN {X 0,Y 495.897,Z 462.712,A -85,B 0,C 180,E1 -6024.308,E2 -6024.308} C_VEL
LIN {X 0,Y 495.908,Z 462.715,A -85,B 0,C 180,E1 -6027.971,E2 -6027.971} C_VEL
LIN {X 0,Y 495.908,Z 462.997,A -85,B 0,C 180,E1 -6028.326,E2 -6028.326} C_VEL
LIN {X 0,Y 496.219,Z 464.262,A -85,B 0,C 180,E1 -6028.446,E2 -6028.446} C_VEL
LIN {X 0,Y 498.664,Z 471.544,A -85,B 0,C 180,E1 -6028.639,E2 -6028.639} C_VEL
LIN {X 0,Y 498.285,Z 543.348,A -85,B 0,C 180,E1 -6029.698,E2 -6029.698} C_VEL
LIN {X 0,Y 498.185,Z 556.42,A -85,B 0,C 180,E1 -6030.052,E2 -6030.052} C_VEL
LIN {X 0,Y 498.055,Z 568.927,A -85,B 0,C 180,E1 -6030.557,E2 -6030.557} C_VEL
LIN {X 0,Y 497.789,Z 580.941,A -85,B 0,C 180,E1 -6031.215,E2 -6031.215} C_VEL
LIN {X 0,Y 497.485,Z 592.288,A -85,B 0,C 180,E1 -6032.025,E2 -6032.025} C_VEL
LIN {X 0,Y 497.104,Z 602.542,A -85,B 0,C 180,E1 -6032.939,E2 -6032.939} C_VEL
LIN {X 0,Y 496.841,Z 610.91,A -85,B 0,C 180,E1 -6033.854,E2 -6033.854} C_VEL
LIN {X 0,Y 496.549,Z 618.65,A -85,B 0,C 180,E1 -6034.873,E2 -6034.873} C_VEL
LIN {X 0,Y 496.321,Z 626.208,A -85,B 0,C 180,E1 -6036.098,E2 -6036.098} C_VEL
LIN {X 0,Y 496.053,Z 632.476,A -85,B 0,C 180,E1 -6037.368,E2 -6037.368} C_VEL
LIN {X 0,Y 495.862,Z 637.138,A -85,B 0,C 180,E1 -6038.56,E2 -6038.56} C_VEL
LIN {X 0,Y 495.698,Z 640.881,A -85,B 0,C 180,E1 -6039.797,E2 -6039.797} C_VEL
LIN {X 0,Y 495.606,Z 642.815,A -85,B 0,C 180,E1 -6040.624,E2 -6040.624} C_VEL
LIN {X 0,Y 495.548,Z 644.912,A -85,B 0,C 180,E1 -6041.883,E2 -6041.883} C_VEL
LIN {X 0,Y 495.504,Z 646.049,A -85,B 0,C 180,E1 -6043.118,E2 -6043.118} C_VEL
LIN {X 0,Y 495.481,Z 646.333,A -85,B 0,C 180,E1 -6043.955,E2 -6043.955} C_VEL
LIN {X 0,Y 495.536,Z 645.883,A -85,B 0,C 180,E1 -6045.331,E2 -6045.331} C_VEL
LIN {X 0,Y 495.568,Z 644.638,A -85,B 0,C 180,E1 -6046.478,E2 -6046.478} C_VEL
LIN {X 0,Y 495.613,Z 643.242,A -85,B 0,C 180,E1 -6047.326,E2 -6047.326} C_VEL
LIN {X 0,Y 495.744,Z 640.371,A -85,B 0,C 180,E1 -6048.559,E2 -6048.559} C_VEL
LIN {X 0,Y 495.95,Z 636.12,A -85,B 0,C 180,E1 -6049.884,E2 -6049.884} C_VEL
LIN {X 0,Y 496.209,Z 629.671,A -85,B 0,C 180,E1 -6051.391,E2 -6051.391} C_VEL
LIN {X 0,Y 496.431,Z 623.799,A -85,B 0,C 180,E1 -6052.474,E2 -6052.474} C_VEL
LIN {X 0,Y 496.733,Z 616.64,A -85,B 0,C 180,E1 -6053.56,E2 -6053.56} C_VEL
LIN {X 0,Y 497.066,Z 607.85,A -85,B 0,C 180,E1 -6054.653,E2 -6054.653} C_VEL
LIN {X 0,Y 497.403,Z 597.931,A -85,B 0,C 180,E1 -6055.646,E2 -6055.646} C_VEL
LIN {X 0,Y 497.752,Z 587.037,A -85,B 0,C 180,E1 -6056.522,E2 -6056.522} C_VEL
LIN {X 0,Y 498.074,Z 575.378,A -85,B 0,C 180,E1 -6057.259,E2 -6057.259} C_VEL
LIN {X 0,Y 498.251,Z 562.767,A -85,B 0,C 180,E1 -6057.856,E2 -6057.856} C_VEL
LIN {X 0,Y 498.37,Z 550.164,A -85,B 0,C 180,E1 -6058.278,E2 -6058.278} C_VEL
LIN {X 0,Y 498.399,Z 537.767,A -85,B 0,C 180,E1 -6058.535,E2 -6058.535} C_VEL
LIN {X 0,Y 498.706,Z 471.122,A -85,B 0,C 180,E1 -6059.513,E2 -6059.513} C_VEL
LIN {X 0,Y 495.959,Z 463.61,A -85,B 0,C 180,E1 -6059.748,E2 -6059.748} C_VEL
LIN {X 0,Y 495.791,Z 462.785,A -85,B 0,C 180,E1 -6059.927,E2 -6059.927} C_VEL
LIN {X 0,Y 495.792,Z 462.727,A -85,B 0,C 180,E1 -6063.245,E2 -6063.245} C_VEL
LIN {X 0,Y 495.723,Z 462.734,A -85,B 0,C 180,E1 -6066.089,E2 -6066.089} C_VEL
LIN {X 0,Y 495.767,Z 462.732,A -85,B 0,C 180,E1 -6068.769,E2 -6068.769} C_VEL
LIN {X 0,Y 495.76,Z 462.726,A -85,B 0,C 180,E1 -6071.782,E2 -6071.782} C_VEL
LIN {X 0,Y 495.741,Z 462.735,A -85,B 0,C 180,E1 -6075.142,E2 -6075.142} C_VEL
LIN {X 0,Y 495.76,Z 462.73,A -85,B 0,C 180,E1 -6078.22,E2 -6078.22} C_VEL
LIN {X 0,Y 495.754,Z 462.731,A -85,B 0,C 180,E1 -6081.409,E2 -6081.409} C_VEL
LIN {X 0,Y 495.784,Z 462.922,A -85,B 0,C 180,E1 -6082.251,E2 -6082.251} C_VEL
LIN {X 0,Y 497.682,Z 472.586,A -85,B 0,C 180,E1 -6083.892,E2 -6083.892} C_VEL
LIN {X 0,Y 497.446,Z 486.401,A -85,B 0,C 180,E1 -6086.079,E2 -6086.079} C_VEL
LIN {X 0,Y 496.988,Z 504.363,A -85,B 0,C 180,E1 -6088.926,E2 -6088.926} C_VEL
LIN {X 0,Y 496.703,Z 517.865,A -85,B 0,C 180,E1 -6091.023,E2 -6091.023} C_VEL
LIN {X 0,Y 498.618,Z 529.591,A -85,B 0,C 180,E1 -6091.294,E2 -6091.294} C_VEL
LIN {X 0,Y 497.899,Z 626.412,A -85,B 0,C 180,E1 -6092.767,E2 -6092.767} C_VEL
LIN {X 0,Y 497.638,Z 639.843,A -85,B 0,C 180,E1 -6093.133,E2 -6093.133} C_VEL
LIN {X 0,Y 497.318,Z 652.976,A -85,B 0,C 180,E1 -6093.68,E2 -6093.68} C_VEL
LIN {X 0,Y 497.006,Z 664.733,A -85,B 0,C 180,E1 -6094.339,E2 -6094.339} C_VEL
LIN {X 0,Y 496.682,Z 675.409,A -85,B 0,C 180,E1 -6095.105,E2 -6095.105} C_VEL
LIN {X 0,Y 496.252,Z 686.305,A -85,B 0,C 180,E1 -6096.085,E2 -6096.085} C_VEL
LIN {X 0,Y 495.944,Z 695.387,A -85,B 0,C 180,E1 -6097.091,E2 -6097.091} C_VEL
LIN {X 0,Y 495.686,Z 703.212,A -85,B 0,C 180,E1 -6098.15,E2 -6098.15} C_VEL
LIN {X 0,Y 495.403,Z 710.922,A -85,B 0,C 180,E1 -6099.442,E2 -6099.442} C_VEL
LIN {X 0,Y 495.29,Z 716.128,A -85,B 0,C 180,E1 -6100.522,E2 -6100.522} C_VEL
LIN {X 0,Y 495.146,Z 721.695,A -85,B 0,C 180,E1 -6101.989,E2 -6101.989} C_VEL
LIN {X 0,Y 495.003,Z 725.759,A -85,B 0,C 180,E1 -6103.504,E2 -6103.504} C_VEL
LIN {X 0,Y 494.961,Z 728.221,A -85,B 0,C 180,E1 -6104.918,E2 -6104.918} C_VEL
LIN {X 0,Y 494.941,Z 729.285,A -85,B 0,C 180,E1 -6106.031,E2 -6106.031} C_VEL
LIN {X 0,Y 494.935,Z 729.599,A -85,B 0,C 180,E1 -6106.868,E2 -6106.868} C_VEL
LIN {X 0,Y 495.029,Z 729.066,A -85,B 0,C 180,E1 -6108.412,E2 -6108.412} C_VEL
LIN {X 0,Y 495.038,Z 728.01,A -85,B 0,C 180,E1 -6109.365,E2 -6109.365} C_VEL
LIN {X 0,Y 494.995,Z 726.672,A -85,B 0,C 180,E1 -6110.191,E2 -6110.191} C_VEL
LIN {X 0,Y 495.11,Z 723.805,A -85,B 0,C 180,E1 -6111.429,E2 -6111.429} C_VEL
LIN {X 0,Y 495.221,Z 719.901,A -85,B 0,C 180,E1 -6112.662,E2 -6112.662} C_VEL
LIN {X 0,Y 495.335,Z 714.844,A -85,B 0,C 180,E1 -6113.892,E2 -6113.892} C_VEL
LIN {X 0,Y 495.46,Z 708.487,A -85,B 0,C 180,E1 -6115.118,E2 -6115.118} C_VEL
LIN {X 0,Y 495.738,Z 700.589,A -85,B 0,C 180,E1 -6116.343,E2 -6116.343} C_VEL
LIN {X 0,Y 496.085,Z 692.517,A -85,B 0,C 180,E1 -6117.361,E2 -6117.361} C_VEL
LIN {X 0,Y 496.385,Z 682.634,A -85,B 0,C 180,E1 -6118.378,E2 -6118.378} C_VEL
LIN {X 0,Y 496.789,Z 671.557,A -85,B 0,C 180,E1 -6119.291,E2 -6119.291} C_VEL
LIN {X 0,Y 497.131,Z 660.745,A -85,B 0,C 180,E1 -6120,E2 -6120} C_VEL
LIN {X 0,Y 497.454,Z 648.662,A -85,B 0,C 180,E1 -6120.607,E2 -6120.607} C_VEL
LIN {X 0,Y 497.657,Z 635.532,A -85,B 0,C 180,E1 -6121.088,E2 -6121.088} C_VEL
LIN {X 0,Y 497.878,Z 622.199,A -85,B 0,C 180,E1 -6121.391,E2 -6121.391} C_VEL
LIN {X 0,Y 498.501,Z 528.789,A -85,B 0,C 180,E1 -6122.816,E2 -6122.816} C_VEL
LIN {X 0,Y 496.903,Z 518.95,A -85,B 0,C 180,E1 -6123.041,E2 -6123.041} C_VEL
LIN {X 0,Y 496.843,Z 515.95,A -85,B 0,C 180,E1 -6123.447,E2 -6123.447} C_VEL
LIN {X 0,Y 497.239,Z 497.798,A -85,B 0,C 180,E1 -6126.289,E2 -6126.289} C_VEL
LIN {X 0,Y 497.587,Z 477.803,A -85,B 0,C 180,E1 -6129.348,E2 -6129.348} C_VEL
LIN {X 0,Y 497.584,Z 472.395,A -85,B 0,C 180,E1 -6130.169,E2 -6130.169} C_VEL
LIN {X 0,Y 495.89,Z 462.823,A -85,B 0,C 180,E1 -6131.716,E2 -6131.716} C_VEL
LIN {X 0,Y 495.831,Z 462.725,A -85,B 0,C 180,E1 -6135.451,E2 -6135.451} C_VEL
LIN {X 0,Y 495.785,Z 462.731,A -85,B 0,C 180,E1 -6139.029,E2 -6139.029} C_VEL
LIN {X 0,Y 495.749,Z 462.731,A -85,B 0,C 180,E1 -6141.629,E2 -6141.629} C_VEL
LIN {X 0,Y 495.724,Z 462.734,A -85,B 0,C 180,E1 -6144.277,E2 -6144.277} C_VEL
LIN {X 0,Y 495.792,Z 462.73,A -85,B 0,C 180,E1 -6146.976,E2 -6146.976} C_VEL
LIN {X 0,Y 495.774,Z 462.726,A -85,B 0,C 180,E1 -6149.746,E2 -6149.746} C_VEL
LIN {X 0,Y 495.776,Z 462.73,A -85,B 0,C 180,E1 -6152.594,E2 -6152.594} C_VEL
LIN {X 0,Y 495.756,Z 462.728,A -85,B 0,C 180,E1 -6155.537,E2 -6155.537} C_VEL
LIN {X 0,Y 495.771,Z 462.732,A -85,B 0,C 180,E1 -6158.768,E2 -6158.768} C_VEL
LIN {X 0,Y 495.764,Z 462.728,A -85,B 0,C 180,E1 -6161.781,E2 -6161.781} C_VEL
LIN {X 0,Y 495.745,Z 462.731,A -85,B 0,C 180,E1 -6165.14,E2 -6165.14} C_VEL
LIN {X 0,Y 495.764,Z 462.733,A -85,B 0,C 180,E1 -6168.218,E2 -6168.218} C_VEL
LIN {X 0,Y 495.754,Z 462.72,A -85,B 0,C 180,E1 -6171.407,E2 -6171.407} C_VEL
LIN {X 0,Y 495.75,Z 462.73,A -85,B 0,C 180,E1 -6174.461,E2 -6174.461} C_VEL
LIN {X 0,Y 495.759,Z 462.732,A -85,B 0,C 180,E1 -6177.404,E2 -6177.404} C_VEL
LIN {X 0,Y 495.845,Z 462.952,A -85,B 0,C 180,E1 -6180.593,E2 -6180.593} C_VEL
LIN {X 0,Y 498.828,Z 476.646,A -85,B 0,C 180,E1 -6182.575,E2 -6182.575} C_VEL
LIN {X 0,Y 498.902,Z 483.182,A -85,B 0,C 180,E1 -6183.431,E2 -6183.431} C_VEL
LIN {X 0,Y 498.017,Z 509.233,A -85,B 0,C 180,E1 -6186.724,E2 -6186.724} C_VEL
LIN {X 0,Y 497.299,Z 533.604,A -85,B 0,C 180,E1 -6189.741,E2 -6189.741} C_VEL
LIN {X 0,Y 496.674,Z 557.929,A -85,B 0,C 180,E1 -6192.712,E2 -6192.712} C_VEL
LIN {X 0,Y 496.456,Z 568.218,A -85,B 0,C 180,E1 -6193.932,E2 -6193.932} C_VEL
LIN {X 0,Y 498.46,Z 586.416,A -85,B 0,C 180,E1 -6194.276,E2 -6194.276} C_VEL
LIN {X 0,Y 497.919,Z 678.45,A -85,B 0,C 180,E1 -6195.62,E2 -6195.62} C_VEL
LIN {X 0,Y 497.543,Z 691.899,A -85,B 0,C 180,E1 -6195.974,E2 -6195.974} C_VEL
LIN {X 0,Y 497.185,Z 705.36,A -85,B 0,C 180,E1 -6196.511,E2 -6196.511} C_VEL
LIN {X 0,Y 496.854,Z 716.955,A -85,B 0,C 180,E1 -6197.143,E2 -6197.143} C_VEL
LIN {X 0,Y 496.498,Z 728.475,A -85,B 0,C 180,E1 -6197.947,E2 -6197.947} C_VEL
LIN {X 0,Y 496.032,Z 739.09,A -85,B 0,C 180,E1 -6198.868,E2 -6198.868} C_VEL
LIN {X 0,Y 495.804,Z 747.813,A -85,B 0,C 180,E1 -6199.793,E2 -6199.793} C_VEL
LIN {X 0,Y 495.578,Z 755.874,A -85,B 0,C 180,E1 -6200.818,E2 -6200.818} C_VEL
LIN {X 0,Y 495.367,Z 763.764,A -85,B 0,C 180,E1 -6202.048,E2 -6202.048} C_VEL
LIN {X 0,Y 495.212,Z 770.832,A -85,B 0,C 180,E1 -6203.432,E2 -6203.432} C_VEL
LIN {X 0,Y 495.196,Z 775.907,A -85,B 0,C 180,E1 -6204.706,E2 -6204.706} C_VEL
LIN {X 0,Y 495.207,Z 779.646,A -85,B 0,C 180,E1 -6205.93,E2 -6205.93} C_VEL
LIN {X 0,Y 495.153,Z 781.531,A -85,B 0,C 180,E1 -6206.744,E2 -6206.744} C_VEL
LIN {X 0,Y 495.135,Z 782.991,A -85,B 0,C 180,E1 -6207.558,E2 -6207.558} C_VEL
LIN {X 0,Y 495.086,Z 784.027,A -85,B 0,C 180,E1 -6208.372,E2 -6208.372} C_VEL
LIN {X 0,Y 495.06,Z 784.655,A -85,B 0,C 180,E1 -6209.185,E2 -6209.185} C_VEL
LIN {X 0,Y 495.121,Z 784.883,A -85,B 0,C 180,E1 -6209.999,E2 -6209.999} C_VEL
LIN {X 0,Y 495.081,Z 784.065,A -85,B 0,C 180,E1 -6211.626,E2 -6211.626} C_VEL
LIN {X 0,Y 495.129,Z 783.044,A -85,B 0,C 180,E1 -6212.439,E2 -6212.439} C_VEL
LIN {X 0,Y 495.147,Z 781.596,A -85,B 0,C 180,E1 -6213.253,E2 -6213.253} C_VEL
LIN {X 0,Y 495.138,Z 778.547,A -85,B 0,C 180,E1 -6214.476,E2 -6214.476} C_VEL
LIN {X 0,Y 495.227,Z 774.516,A -85,B 0,C 180,E1 -6215.7,E2 -6215.7} C_VEL
LIN {X 0,Y 495.27,Z 768.372,A -85,B 0,C 180,E1 -6217.111,E2 -6217.111} C_VEL
LIN {X 0,Y 495.44,Z 761.447,A -85,B 0,C 180,E1 -6218.359,E2 -6218.359} C_VEL
LIN {X 0,Y 495.638,Z 752.968,A -85,B 0,C 180,E1 -6219.589,E2 -6219.589} C_VEL
LIN {X 0,Y 495.918,Z 744.32,A -85,B 0,C 180,E1 -6220.615,E2 -6220.615} C_VEL
LIN {X 0,Y 496.269,Z 733.659,A -85,B 0,C 180,E1 -6221.641,E2 -6221.641} C_VEL
LIN {X 0,Y 496.691,Z 722.061,A -85,B 0,C 180,E1 -6222.538,E2 -6222.538} C_VEL
LIN {X 0,Y 497.034,Z 709.673,A -85,B 0,C 180,E1 -6223.282,E2 -6223.282} C_VEL
LIN {X 0,Y 497.454,Z 697.216,A -85,B 0,C 180,E1 -6223.843,E2 -6223.843} C_VEL
LIN {X 0,Y 497.741,Z 684.439,A -85,B 0,C 180,E1 -6224.252,E2 -6224.252} C_VEL
LIN {X 0,Y 497.989,Z 671.084,A -85,B 0,C 180,E1 -6224.506,E2 -6224.506} C_VEL
LIN {X 0,Y 498.374,Z 585.125,A -85,B 0,C 180,E1 -6225.75,E2 -6225.75} C_VEL
LIN {X 0,Y 496.471,Z 568.4,A -85,B 0,C 180,E1 -6226.077,E2 -6226.077} C_VEL
LIN {X 0,Y 497.018,Z 544.52,A -85,B 0,C 180,E1 -6228.978,E2 -6228.978} C_VEL
LIN {X 0,Y 497.77,Z 518.532,A -85,B 0,C 180,E1 -6232.189,E2 -6232.189} C_VEL
LIN {X 0,Y 498.515,Z 495.939,A -85,B 0,C 180,E1 -6235.018,E2 -6235.018} C_VEL
LIN {X 0,Y 499.072,Z 478.08,A -85,B 0,C 180,E1 -6237.285,E2 -6237.285} C_VEL
LIN {X 0,Y 495.82,Z 462.858,A -85,B 0,C 180,E1 -6239.449,E2 -6239.449} C_VEL
LIN {X 0,Y 495.761,Z 462.732,A -85,B 0,C 180,E1 -6242.593,E2 -6242.593} C_VEL
LIN {X 0,Y 495.735,Z 462.733,A -85,B 0,C 180,E1 -6245.537,E2 -6245.537} C_VEL
LIN {X 0,Y 495.733,Z 462.731,A -85,B 0,C 180,E1 -6248.763,E2 -6248.763} C_VEL
LIN {X 0,Y 495.735,Z 462.732,A -85,B 0,C 180,E1 -6251.781,E2 -6251.781} C_VEL
LIN {X 0,Y 495.728,Z 462.73,A -85,B 0,C 180,E1 -6255.139,E2 -6255.139} C_VEL
LIN {X 0,Y 495.735,Z 462.738,A -85,B 0,C 180,E1 -6258.216,E2 -6258.216} C_VEL
LIN {X 0,Y 495.735,Z 462.729,A -85,B 0,C 180,E1 -6261.407,E2 -6261.407} C_VEL
LIN {X 0,Y 495.734,Z 462.735,A -85,B 0,C 180,E1 -6264.461,E2 -6264.461} C_VEL
LIN {X 0,Y 495.756,Z 462.726,A -85,B 0,C 180,E1 -6267.404,E2 -6267.404} C_VEL
LIN {X 0,Y 495.754,Z 462.734,A -85,B 0,C 180,E1 -6270.252,E2 -6270.252} C_VEL
LIN {X 0,Y 495.793,Z 462.721,A -85,B 0,C 180,E1 -6273.254,E2 -6273.254} C_VEL
LIN {X 0,Y 495.727,Z 462.735,A -85,B 0,C 180,E1 -6276.611,E2 -6276.611} C_VEL
LIN {X 0,Y 495.765,Z 462.725,A -85,B 0,C 180,E1 -6279.323,E2 -6279.323} C_VEL
LIN {X 0,Y 495.777,Z 462.725,A -85,B 0,C 180,E1 -6281.828,E2 -6281.828} C_VEL
LIN {X 0,Y 495.81,Z 462.727,A -85,B 0,C 180,E1 -6284.548,E2 -6284.548} C_VEL
LIN {X 0,Y 495.816,Z 462.721,A -85,B 0,C 180,E1 -6287.964,E2 -6287.964} C_VEL
LIN {X 0,Y 495.827,Z 462.719,A -85,B 0,C 180,E1 -6291.03,E2 -6291.03} C_VEL
LIN {X 0,Y 495.842,Z 462.715,A -85,B 0,C 180,E1 -6293.489,E2 -6293.489} C_VEL
LIN {X 0,Y 495.829,Z 462.723,A -85,B 0,C 180,E1 -6296.749,E2 -6296.749} C_VEL
LIN {X 0,Y 495.991,Z 462.698,A -85,B 0,C 180,E1 -6299.188,E2 -6299.188} C_VEL
LIN {X 0,Y 495.854,Z 462.714,A -85,B 0,C 180,E1 -6301.624,E2 -6301.624} C_VEL
LIN {X 0,Y 495.829,Z 462.718,A -85,B 0,C 180,E1 -6303.25,E2 -6303.25} C_VEL
LIN {X 0,Y 495.845,Z 462.723,A -85,B 0,C 180,E1 -6306.51,E2 -6306.51} C_VEL
LIN {X 0,Y 495.831,Z 462.721,A -85,B 0,C 180,E1 -6308.97,E2 -6308.97} C_VEL
LIN {X 0,Y 495.796,Z 462.725,A -85,B 0,C 180,E1 -6312.276,E2 -6312.276} C_VEL
LIN {X 0,Y 495.809,Z 462.72,A -85,B 0,C 180,E1 -6315.452,E2 -6315.452} C_VEL
LIN {X 0,Y 495.792,Z 462.725,A -85,B 0,C 180,E1 -6318.248,E2 -6318.248} C_VEL
LIN {X 0,Y 495.76,Z 462.734,A -85,B 0,C 180,E1 -6320.757,E2 -6320.757} C_VEL
LIN {X 0,Y 495.738,Z 462.729,A -85,B 0,C 180,E1 -6323.387,E2 -6323.387} C_VEL
LIN {X 0,Y 495.785,Z 462.723,A -85,B 0,C 180,E1 -6326.068,E2 -6326.068} C_VEL
LIN {X 0,Y 495.759,Z 462.734,A -85,B 0,C 180,E1 -6328.815,E2 -6328.815} C_VEL
LIN {X 0,Y 495.745,Z 462.727,A -85,B 0,C 180,E1 -6331.727,E2 -6331.727} C_VEL
LIN {X 0,Y 495.764,Z 462.733,A -85,B 0,C 180,E1 -6334.696,E2 -6334.696} C_VEL
LIN {X 0,Y 495.719,Z 462.731,A -85,B 0,C 180,E1 -6337.562,E2 -6337.562} C_VEL
LIN {X 0,Y 495.755,Z 462.733,A -85,B 0,C 180,E1 -6340.701,E2 -6340.701} C_VEL
LIN {X 0,Y 495.723,Z 462.73,A -85,B 0,C 180,E1 -6343.696,E2 -6343.696} C_VEL
LIN {X 0,Y 495.724,Z 462.732,A -85,B 0,C 180,E1 -6346.305,E2 -6346.305} C_VEL
LIN {X 0,Y 495.772,Z 462.728,A -85,B 0,C 180,E1 -6349.303,E2 -6349.303} C_VEL
LIN {X 0,Y 495.754,Z 462.729,A -85,B 0,C 180,E1 -6351.411,E2 -6351.411} C_VEL
LIN {X 0,Y 495.746,Z 462.73,A -85,B 0,C 180,E1 -6354.464,E2 -6354.464} C_VEL
LIN {X 0,Y 495.761,Z 462.728,A -85,B 0,C 180,E1 -6357.407,E2 -6357.407} C_VEL
LIN {X 0,Y 495.758,Z 462.726,A -85,B 0,C 180,E1 -6360.255,E2 -6360.255} C_VEL
LIN {X 0,Y 495.746,Z 462.729,A -85,B 0,C 180,E1 -6360.775,E2 -6360.775} C_VEL
LIN {X 0,Y 495.09,Z 462.814,A -85,B 0,C 180,E1 -6361.454,E2 -6361.454} C_VEL
LIN {X 0,Y 492.233,Z 463.168,A -85,B 0,C 180,E1 -6362.556,E2 -6362.556} C_VEL
LIN {X 0,Y 489.823,Z 463.468,A -85,B 0,C 180,E1 -6363.445,E2 -6363.445} C_VEL
LIN {X 0,Y 488.808,Z 463.592,A -85,B 0,C 180,E1 -6364.131,E2 -6364.131} C_VEL
LIN {X 0,Y 488.736,Z 463.602,A -85,B 0,C 180,E1 -6364.363,E2 -6364.363} C_VEL
LIN {X 0,Y 488.715,Z 463.611,A -85,B 0,C 180,E1 -6367.154,E2 -6367.154} C_VEL
LIN {X 0,Y 488.723,Z 463.603,A -85,B 0,C 180,E1 -6369.812,E2 -6369.812} C_VEL
LIN {X 0,Y 488.729,Z 463.602,A -85,B 0,C 180,E1 -6372.425,E2 -6372.425} C_VEL
LIN {X 0,Y 488.758,Z 463.605,A -85,B 0,C 180,E1 -6375.001,E2 -6375.001} C_VEL
LIN {X 0,Y 488.802,Z 463.593,A -85,B 0,C 180,E1 -6378.389,E2 -6378.389} C_VEL
LIN {X 0,Y 488.815,Z 463.595,A -85,B 0,C 180,E1 -6381.735,E2 -6381.735} C_VEL
LIN {X 0,Y 488.856,Z 463.59,A -85,B 0,C 180,E1 -6384.226,E2 -6384.226} C_VEL
LIN {X 0,Y 488.892,Z 463.607,A -85,B 0,C 180,E1 -6387.942,E2 -6387.942} C_VEL
LIN {X 0,Y 488.927,Z 464.055,A -85,B 0,C 180,E1 -6388.148,E2 -6388.148} C_VEL
LIN {X 0,Y 489.359,Z 465.636,A -85,B 0,C 180,E1 -6388.246,E2 -6388.246} C_VEL
LIN {X 0,Y 491.838,Z 472.976,A -85,B 0,C 180,E1 -6388.441,E2 -6388.441} C_VEL
